(* CODESYS project 0427直角+Delta.project
   CompiledLibraryCompatibilityVersion: LeadSysStudio V3.5 SP15 Patch 4
   Title: Untitled2

Project tree, tasks and I/O mapping:
  Device : PMC600, Leadshine Technology Co., Ltd., order no. 600101, version 3.5.15.40
    application Application
      libraries: Standard, * (System)
      task MainTask (cyclic, interval t#4ms, priority 4, watchdog t#5000ms x 1) calls nothing
      task EtherCAT_Master_Leadshine_A (cyclic, interval 4000 µs, priority 0) calls PLC_PRG, EtherCAT_Master_Leadshine_A.EtherCAT_Task
      task SoftMotion_PlanningTask (freewheeling, priority 15) calls nothing
      program PLC_PRG [LD]
      axis group Tripod: TRAFO.Kin_Tripod_Rotary, axes Axis_3, Axis_4, Axis_5
    Device Diagnose
    Network Configuration
      LocalBus Config
    Resource Usage
    SoftMotion General Axis Pool
    High_Speed_IO_Module : High Speed IO Module, Leadshine Technology Co., Ltd., version 3.5.15.40
        settings: HS counter 2.Counter_Channel = 1; HS counter 3.Counter_Channel = 2; HS counter 4.Counter_Channel = 3; HS counter 5.Counter_Channel = 4; HS counter 6.Counter_Channel = 5
        unmapped channels: Genral_IO_IN, Genral_IO_Out
    EtherCAT_Master_Leadshine_A : EtherCAT Master Leadshine, Leadshine Technology Co., Ltd., version 3.5.9.50
        settings: MasterCycleTime = 4000
      PM32EC_LOCAL : PM32EC-LOCAL, Leadshine Technology Co., Ltd., order no. PM32EC-LOCAL, version Revision=16#20061010
          settings: StationAlias = 0; DC sync0 cycletime = 4000; DC sync1 cycletime = 4000
      DM3C_EC522 : DM3C-EC522(COE), Leadshine Technology Co.,Ltd., order no. DM3C-EC522, version Revision=16#00000001
          settings: StationAlias = 0; DC sync0 cycletime = 4000; DC sync1 cycletime = 4000; Number of SDO = 6; Homing method.Index = 16#6098; Homing method.Subindex = 16#00; Homing method.Value = 17; Homing method.Size = 8; Homing method.AbortIfError = FALSE; Homing method.JumpToLine = FALSE; Homing method.Line = 0; Homing method.CompleteAccess = FALSE; Homing velocity (fast).Index = 16#6099; Homing velocity (fast).Subindex = 16#01; Homing velocity (fast).Value = 16667; Homing velocity (fast).Size = 32; Homing velocity (fast).AbortIfError = FALSE; Homing velocity (fast).JumpToLine = FALSE; Homing velocity (fast).Line = 0; Homing velocity (fast).CompleteAccess = FALSE; Homing velocity (slow).Index = 16#6099; Homing velocity (slow).Subindex = 16#02; Homing velocity (slow).Value = 3333; Homing velocity (slow).Size = 32; Homing velocity (slow).AbortIfError = FALSE; Homing velocity (slow).JumpToLine = FALSE; Homing velocity (slow).Line = 0; Homing velocity (slow).CompleteAccess = FALSE; Homing acceleration.Index = 16#609A; Homing acceleration.Subindex = 16#00; Homing acceleration.Value = 83333; Homing acceleration.Size = 32; Homing acceleration.AbortIfError = FALSE; Homing acceleration.JumpToLine = FALSE; Homing acceleration.Line = 0; Homing acceleration.CompleteAccess = FALSE; Homing offset.Index = 16#607C; Homing offset.Subindex = 16#00; Homing offset.Value = 0; Homing offset.Size = 32;
            Homing offset.AbortIfError = FALSE; Homing offset.JumpToLine = FALSE; Homing offset.Line = 0; Homing offset.CompleteAccess = FALSE
          unmapped channels: Control Word, Profile Target Position, Touch Probe Function, Last Error Code, Status Word, Modes of Operation display, Position Actual Value, Touch Probe Status, Touch Probe 1 Positive Value, Digital Inputs
        Axis : Axis, 3S - Smart Software Solutions GmbH, order no. 0, version 4.6.1.0
            settings: wDriveID = 0; dwRatioTechUnitsDenom = 2500; iRatioTechUnitsNum = 3; 一圈脉冲数 = 50000; 工作台一圈的位移 = 60; 电子齿轮比分子 = 1; 电子齿轮比分母 = 1; ScalingIncs = 2500; ScalingUnits = 3; AdrOffset_8010 = 4; BitOffset_8010 = 0; BitLength_8010 = 16; Address_8010 = '%QW2'; Type_8010 = 'UINT'; AddressPointer_8010 = ADR(%QW2); AdrOffset_8020 = 8; BitOffset_8020 = 0; BitLength_8020 = 32; Address_8020 = '%QD2'; Type_8020 = 'DINT'; AddressPointer_8020 = ADR(%QD2); AdrOffset_8030 = 4294967295; BitOffset_8030 = 0; BitLength_8030 = 32; Address_8030 = ''; Type_8030 = 'DINT'; AddressPointer_8030 = 0; AdrOffset_8040 = 4294967295; BitOffset_8040 = 0; BitLength_8040 = 0; Address_8040 = ''; Type_8040 = ''; AddressPointer_8040 = 0; AdrOffset_8050 = 4294967295; BitOffset_8050 = 0; BitLength_8050 = 8; Address_8050 = ''; Type_8050 = 'USINT'; AddressPointer_8050 = 0; AdrOffset_8060 = 12;
              BitOffset_8060 = 0; BitLength_8060 = 16; Address_8060 = '%QW6'; Type_8060 = 'UINT'; AddressPointer_8060 = ADR(%QW6); AdrOffset_8070 = 4294967295; BitOffset_8070 = 0; BitLength_8070 = 0; Address_8070 = ''; Type_8070 = ''; AddressPointer_8070 = 0; AdrOffset_8080 = 4294967295; BitOffset_8080 = 0; BitLength_8080 = 0; Address_8080 = ''; Type_8080 = ''; AddressPointer_8080 = 0; AdrOffset_8090 = 4294967295; BitOffset_8090 = 0; BitLength_8090 = 0; Address_8090 = ''; Type_8090 = ''; AddressPointer_8090 = 0; AdrOffset_8510 = 6; BitOffset_8510 = 0; BitLength_8510 = 16; Address_8510 = '%IW3'; Type_8510 = 'UINT'; AddressPointer_8510 = ADR(%IW3); AdrOffset_8520 = 12; BitOffset_8520 = 0; BitLength_8520 = 32; Address_8520 = '%ID3'; Type_8520 = 'DINT'; AddressPointer_8520 = ADR(%ID3); AdrOffset_8530 = 4294967295; BitOffset_8530 = 0; BitLength_8530 = 0; Address_8530 = ''; Type_8530 = '';
              AddressPointer_8530 = 0; AdrOffset_8540 = 4294967295; BitOffset_8540 = 0; BitLength_8540 = 0; Address_8540 = ''; Type_8540 = ''; AddressPointer_8540 = 0; AdrOffset_8550 = 8; BitOffset_8550 = 0; BitLength_8550 = 8; Address_8550 = '%IB8'; Type_8550 = 'SINT'; AddressPointer_8550 = ADR(%IB8); AdrOffset_8560 = 24; BitOffset_8560 = 0; BitLength_8560 = 32; Address_8560 = '%ID6'; Type_8560 = 'UDINT'; AddressPointer_8560 = ADR(%ID6); AdrOffset_8570 = 16; BitOffset_8570 = 0; BitLength_8570 = 16; Address_8570 = '%IW8'; Type_8570 = 'UINT'; AddressPointer_8570 = ADR(%IW8); AdrOffset_8580 = 20; BitOffset_8580 = 0; BitLength_8580 = 32; Address_8580 = '%ID5'; Type_8580 = 'DINT'; AddressPointer_8580 = ADR(%ID5); AdrOffset_8590 = 4294967295; BitOffset_8590 = 0; BitLength_8590 = 0; Address_8590 = ''; Type_8590 = ''; AddressPointer_8590 = 0; AdrOffset_8600 = 4294967295; BitOffset_8600 = 0; BitLength_8600 = 0;
              Address_8600 = ''; Type_8600 = ''; AddressPointer_8600 = 0; AdrOffset_8600 = 4294967295; BitOffset_8600 = 0; BitLength_8600 = 0; Address_8610 = ''; Type_8610 = ''; AddressPointer_8610 = 0; AdrOffset_8620 = 4294967295; BitOffset_8620 = 0; BitLength_8620 = 0; Address_8620 = ''; Type_8620 = ''; AddressPointer_8620 = 0
      DM3C_EC522_1 : DM3C-EC522(COE), Leadshine Technology Co.,Ltd., order no. DM3C-EC522, version Revision=16#00000001
          settings: StationAlias = 0; DC sync0 cycletime = 4000; DC sync1 cycletime = 4000; Number of SDO = 6; Homing method.Index = 16#6098; Homing method.Subindex = 16#00; Homing method.Value = 17; Homing method.Size = 8; Homing method.AbortIfError = FALSE; Homing method.JumpToLine = FALSE; Homing method.Line = 0; Homing method.CompleteAccess = FALSE; Homing velocity (fast).Index = 16#6099; Homing velocity (fast).Subindex = 16#01; Homing velocity (fast).Value = 16667; Homing velocity (fast).Size = 32; Homing velocity (fast).AbortIfError = FALSE; Homing velocity (fast).JumpToLine = FALSE; Homing velocity (fast).Line = 0; Homing velocity (fast).CompleteAccess = FALSE; Homing velocity (slow).Index = 16#6099; Homing velocity (slow).Subindex = 16#02; Homing velocity (slow).Value = 3333; Homing velocity (slow).Size = 32; Homing velocity (slow).AbortIfError = FALSE; Homing velocity (slow).JumpToLine = FALSE; Homing velocity (slow).Line = 0; Homing velocity (slow).CompleteAccess = FALSE; Homing acceleration.Index = 16#609A; Homing acceleration.Subindex = 16#00; Homing acceleration.Value = 83333; Homing acceleration.Size = 32; Homing acceleration.AbortIfError = FALSE; Homing acceleration.JumpToLine = FALSE; Homing acceleration.Line = 0; Homing acceleration.CompleteAccess = FALSE; Homing offset.Index = 16#607C; Homing offset.Subindex = 16#00; Homing offset.Value = 0; Homing offset.Size = 32;
            Homing offset.AbortIfError = FALSE; Homing offset.JumpToLine = FALSE; Homing offset.Line = 0; Homing offset.CompleteAccess = FALSE
          unmapped channels: Control Word, Profile Target Position, Touch Probe Function, Last Error Code, Status Word, Modes of Operation display, Position Actual Value, Touch Probe Status, Touch Probe 1 Positive Value, Digital Inputs
        Axis_1 : Axis, 3S - Smart Software Solutions GmbH, order no. 0, version 4.6.1.0
            settings: dwRatioTechUnitsDenom = 2500; iRatioTechUnitsNum = 3; 一圈脉冲数 = 50000; 工作台一圈的位移 = 60; 电子齿轮比分子 = 1; 电子齿轮比分母 = 1; ScalingIncs = 2500; ScalingUnits = 3; AdrOffset_8010 = 16; BitOffset_8010 = 0; BitLength_8010 = 16; Address_8010 = '%QW8'; Type_8010 = 'UINT'; AddressPointer_8010 = ADR(%QW8); AdrOffset_8020 = 20; BitOffset_8020 = 0; BitLength_8020 = 32; Address_8020 = '%QD5'; Type_8020 = 'DINT'; AddressPointer_8020 = ADR(%QD5); AdrOffset_8030 = 4294967295; BitOffset_8030 = 0; BitLength_8030 = 32; Address_8030 = ''; Type_8030 = 'DINT'; AddressPointer_8030 = 0; AdrOffset_8040 = 4294967295; BitOffset_8040 = 0; BitLength_8040 = 0; Address_8040 = ''; Type_8040 = ''; AddressPointer_8040 = 0; AdrOffset_8050 = 4294967295; BitOffset_8050 = 0; BitLength_8050 = 8; Address_8050 = ''; Type_8050 = 'USINT'; AddressPointer_8050 = 0; AdrOffset_8060 = 24; BitOffset_8060 = 0;
              BitLength_8060 = 16; Address_8060 = '%QW12'; Type_8060 = 'UINT'; AddressPointer_8060 = ADR(%QW12); AdrOffset_8070 = 4294967295; BitOffset_8070 = 0; BitLength_8070 = 0; Address_8070 = ''; Type_8070 = ''; AddressPointer_8070 = 0; AdrOffset_8080 = 4294967295; BitOffset_8080 = 0; BitLength_8080 = 0; Address_8080 = ''; Type_8080 = ''; AddressPointer_8080 = 0; AdrOffset_8090 = 4294967295; BitOffset_8090 = 0; BitLength_8090 = 0; Address_8090 = ''; Type_8090 = ''; AddressPointer_8090 = 0; AdrOffset_8510 = 30; BitOffset_8510 = 0; BitLength_8510 = 16; Address_8510 = '%IW15'; Type_8510 = 'UINT'; AddressPointer_8510 = ADR(%IW15); AdrOffset_8520 = 36; BitOffset_8520 = 0; BitLength_8520 = 32; Address_8520 = '%ID9'; Type_8520 = 'DINT'; AddressPointer_8520 = ADR(%ID9); AdrOffset_8530 = 4294967295; BitOffset_8530 = 0; BitLength_8530 = 0; Address_8530 = ''; Type_8530 = ''; AddressPointer_8530 = 0;
              AdrOffset_8540 = 4294967295; BitOffset_8540 = 0; BitLength_8540 = 0; Address_8540 = ''; Type_8540 = ''; AddressPointer_8540 = 0; AdrOffset_8550 = 32; BitOffset_8550 = 0; BitLength_8550 = 8; Address_8550 = '%IB32'; Type_8550 = 'SINT'; AddressPointer_8550 = ADR(%IB32); AdrOffset_8560 = 48; BitOffset_8560 = 0; BitLength_8560 = 32; Address_8560 = '%ID12'; Type_8560 = 'UDINT'; AddressPointer_8560 = ADR(%ID12); AdrOffset_8570 = 40; BitOffset_8570 = 0; BitLength_8570 = 16; Address_8570 = '%IW20'; Type_8570 = 'UINT'; AddressPointer_8570 = ADR(%IW20); AdrOffset_8580 = 44; BitOffset_8580 = 0; BitLength_8580 = 32; Address_8580 = '%ID11'; Type_8580 = 'DINT'; AddressPointer_8580 = ADR(%ID11); AdrOffset_8590 = 4294967295; BitOffset_8590 = 0; BitLength_8590 = 0; Address_8590 = ''; Type_8590 = ''; AddressPointer_8590 = 0; AdrOffset_8600 = 4294967295; BitOffset_8600 = 0; BitLength_8600 = 0; Address_8600 = '';
              Type_8600 = ''; AddressPointer_8600 = 0; AdrOffset_8600 = 4294967295; BitOffset_8600 = 0; BitLength_8600 = 0; Address_8610 = ''; Type_8610 = ''; AddressPointer_8610 = 0; AdrOffset_8620 = 4294967295; BitOffset_8620 = 0; BitLength_8620 = 0; Address_8620 = ''; Type_8620 = ''; AddressPointer_8620 = 0
      DM3C_EC522_2 : DM3C-EC522(COE), Leadshine Technology Co.,Ltd., order no. DM3C-EC522, version Revision=16#00000001
          settings: StationAlias = 0; DC sync0 cycletime = 4000; DC sync1 cycletime = 4000; Number of SDO = 6; Homing method.Index = 16#6098; Homing method.Subindex = 16#00; Homing method.Value = 17; Homing method.Size = 8; Homing method.AbortIfError = FALSE; Homing method.JumpToLine = FALSE; Homing method.Line = 0; Homing method.CompleteAccess = FALSE; Homing velocity (fast).Index = 16#6099; Homing velocity (fast).Subindex = 16#01; Homing velocity (fast).Value = 125000; Homing velocity (fast).Size = 32; Homing velocity (fast).AbortIfError = FALSE; Homing velocity (fast).JumpToLine = FALSE; Homing velocity (fast).Line = 0; Homing velocity (fast).CompleteAccess = FALSE; Homing velocity (slow).Index = 16#6099; Homing velocity (slow).Subindex = 16#02; Homing velocity (slow).Value = 25000; Homing velocity (slow).Size = 32; Homing velocity (slow).AbortIfError = FALSE; Homing velocity (slow).JumpToLine = FALSE; Homing velocity (slow).Line = 0; Homing velocity (slow).CompleteAccess = FALSE; Homing acceleration.Index = 16#609A; Homing acceleration.Subindex = 16#00; Homing acceleration.Value = 1250000; Homing acceleration.Size = 32; Homing acceleration.AbortIfError = FALSE; Homing acceleration.JumpToLine = FALSE; Homing acceleration.Line = 0; Homing acceleration.CompleteAccess = FALSE; Homing offset.Index = 16#607C; Homing offset.Subindex = 16#00; Homing offset.Value = 0; Homing offset.Size = 32;
            Homing offset.AbortIfError = FALSE; Homing offset.JumpToLine = FALSE; Homing offset.Line = 0; Homing offset.CompleteAccess = FALSE
          unmapped channels: Control Word, Profile Target Position, Touch Probe Function, Last Error Code, Status Word, Modes of Operation display, Position Actual Value, Touch Probe Status, Touch Probe 1 Positive Value, Digital Inputs
        Axis_2 : Axis, 3S - Smart Software Solutions GmbH, order no. 0, version 4.6.1.0
            settings: wDriveID = 2; dwRatioTechUnitsDenom = 12500; 一圈脉冲数 = 50000; 工作台一圈的位移 = 4; 电子齿轮比分子 = 1; 电子齿轮比分母 = 1; ScalingIncs = 12500; AdrOffset_8010 = 28; BitOffset_8010 = 0; BitLength_8010 = 16; Address_8010 = '%QW14'; Type_8010 = 'UINT'; AddressPointer_8010 = ADR(%QW14); AdrOffset_8020 = 32; BitOffset_8020 = 0; BitLength_8020 = 32; Address_8020 = '%QD8'; Type_8020 = 'DINT'; AddressPointer_8020 = ADR(%QD8); AdrOffset_8030 = 4294967295; BitOffset_8030 = 0; BitLength_8030 = 32; Address_8030 = ''; Type_8030 = 'DINT'; AddressPointer_8030 = 0; AdrOffset_8040 = 4294967295; BitOffset_8040 = 0; BitLength_8040 = 0; Address_8040 = ''; Type_8040 = ''; AddressPointer_8040 = 0; AdrOffset_8050 = 4294967295; BitOffset_8050 = 0; BitLength_8050 = 8; Address_8050 = ''; Type_8050 = 'USINT'; AddressPointer_8050 = 0; AdrOffset_8060 = 36; BitOffset_8060 = 0; BitLength_8060 = 16;
              Address_8060 = '%QW18'; Type_8060 = 'UINT'; AddressPointer_8060 = ADR(%QW18); AdrOffset_8070 = 4294967295; BitOffset_8070 = 0; BitLength_8070 = 0; Address_8070 = ''; Type_8070 = ''; AddressPointer_8070 = 0; AdrOffset_8080 = 4294967295; BitOffset_8080 = 0; BitLength_8080 = 0; Address_8080 = ''; Type_8080 = ''; AddressPointer_8080 = 0; AdrOffset_8090 = 4294967295; BitOffset_8090 = 0; BitLength_8090 = 0; Address_8090 = ''; Type_8090 = ''; AddressPointer_8090 = 0; AdrOffset_8510 = 54; BitOffset_8510 = 0; BitLength_8510 = 16; Address_8510 = '%IW27'; Type_8510 = 'UINT'; AddressPointer_8510 = ADR(%IW27); AdrOffset_8520 = 60; BitOffset_8520 = 0; BitLength_8520 = 32; Address_8520 = '%ID15'; Type_8520 = 'DINT'; AddressPointer_8520 = ADR(%ID15); AdrOffset_8530 = 4294967295; BitOffset_8530 = 0; BitLength_8530 = 0; Address_8530 = ''; Type_8530 = ''; AddressPointer_8530 = 0; AdrOffset_8540 = 4294967295;
              BitOffset_8540 = 0; BitLength_8540 = 0; Address_8540 = ''; Type_8540 = ''; AddressPointer_8540 = 0; AdrOffset_8550 = 56; BitOffset_8550 = 0; BitLength_8550 = 8; Address_8550 = '%IB56'; Type_8550 = 'SINT'; AddressPointer_8550 = ADR(%IB56); AdrOffset_8560 = 72; BitOffset_8560 = 0; BitLength_8560 = 32; Address_8560 = '%ID18'; Type_8560 = 'UDINT'; AddressPointer_8560 = ADR(%ID18); AdrOffset_8570 = 64; BitOffset_8570 = 0; BitLength_8570 = 16; Address_8570 = '%IW32'; Type_8570 = 'UINT'; AddressPointer_8570 = ADR(%IW32); AdrOffset_8580 = 68; BitOffset_8580 = 0; BitLength_8580 = 32; Address_8580 = '%ID17'; Type_8580 = 'DINT'; AddressPointer_8580 = ADR(%ID17); AdrOffset_8590 = 4294967295; BitOffset_8590 = 0; BitLength_8590 = 0; Address_8590 = ''; Type_8590 = ''; AddressPointer_8590 = 0; AdrOffset_8600 = 4294967295; BitOffset_8600 = 0; BitLength_8600 = 0; Address_8600 = ''; Type_8600 = '';
              AddressPointer_8600 = 0; AdrOffset_8600 = 4294967295; BitOffset_8600 = 0; BitLength_8600 = 0; Address_8610 = ''; Type_8610 = ''; AddressPointer_8610 = 0; AdrOffset_8620 = 4294967295; BitOffset_8620 = 0; BitLength_8620 = 0; Address_8620 = ''; Type_8620 = ''; AddressPointer_8620 = 0
      DM3C_EC522_3 : DM3C-EC522(COE), Leadshine Technology Co.,Ltd., order no. DM3C-EC522, version Revision=16#00000001
          settings: StationAlias = 0; DC sync0 cycletime = 4000; DC sync1 cycletime = 4000; Number of SDO = 6; Homing method.Index = 16#6098; Homing method.Subindex = 16#00; Homing method.Value = 21; Homing method.Size = 8; Homing method.AbortIfError = FALSE; Homing method.JumpToLine = FALSE; Homing method.Line = 0; Homing method.CompleteAccess = FALSE; Homing velocity (fast).Index = 16#6099; Homing velocity (fast).Subindex = 16#01; Homing velocity (fast).Value = 7500; Homing velocity (fast).Size = 32; Homing velocity (fast).AbortIfError = FALSE; Homing velocity (fast).JumpToLine = FALSE; Homing velocity (fast).Line = 0; Homing velocity (fast).CompleteAccess = FALSE; Homing velocity (slow).Index = 16#6099; Homing velocity (slow).Subindex = 16#02; Homing velocity (slow).Value = 1500; Homing velocity (slow).Size = 32; Homing velocity (slow).AbortIfError = FALSE; Homing velocity (slow).JumpToLine = FALSE; Homing velocity (slow).Line = 0; Homing velocity (slow).CompleteAccess = FALSE; Homing acceleration.Index = 16#609A; Homing acceleration.Subindex = 16#00; Homing acceleration.Value = 50000; Homing acceleration.Size = 32; Homing acceleration.AbortIfError = FALSE; Homing acceleration.JumpToLine = FALSE; Homing acceleration.Line = 0; Homing acceleration.CompleteAccess = FALSE; Homing offset.Index = 16#607C; Homing offset.Subindex = 16#00; Homing offset.Value = 0; Homing offset.Size = 32;
            Homing offset.AbortIfError = FALSE; Homing offset.JumpToLine = FALSE; Homing offset.Line = 0; Homing offset.CompleteAccess = FALSE
          unmapped channels: Control Word, Profile Target Position, Touch Probe Function, Last Error Code, Status Word, Modes of Operation display, Position Actual Value, Touch Probe Status, Touch Probe 1 Positive Value, Digital Inputs
        Axis_3 : Axis, 3S - Smart Software Solutions GmbH, order no. 0, version 4.6.1.0
            settings: wDriveID = 3; dwRatioTechUnitsDenom = 500; iRatioTechUnitsNum = -1; 一圈脉冲数 = 36000; 工作台一圈的位移 = 360; 电子齿轮比分子 = 5; 电子齿轮比分母 = 1; ScalingIncs = 500; InvertDirection = True; AdrOffset_8010 = 40; BitOffset_8010 = 0; BitLength_8010 = 16; Address_8010 = '%QW20'; Type_8010 = 'UINT'; AddressPointer_8010 = ADR(%QW20); AdrOffset_8020 = 44; BitOffset_8020 = 0; BitLength_8020 = 32; Address_8020 = '%QD11'; Type_8020 = 'DINT'; AddressPointer_8020 = ADR(%QD11); AdrOffset_8030 = 4294967295; BitOffset_8030 = 0; BitLength_8030 = 32; Address_8030 = ''; Type_8030 = 'DINT'; AddressPointer_8030 = 0; AdrOffset_8040 = 4294967295; BitOffset_8040 = 0; BitLength_8040 = 0; Address_8040 = ''; Type_8040 = ''; AddressPointer_8040 = 0; AdrOffset_8050 = 4294967295; BitOffset_8050 = 0; BitLength_8050 = 8; Address_8050 = ''; Type_8050 = 'USINT'; AddressPointer_8050 = 0; AdrOffset_8060 = 48;
              BitOffset_8060 = 0; BitLength_8060 = 16; Address_8060 = '%QW24'; Type_8060 = 'UINT'; AddressPointer_8060 = ADR(%QW24); AdrOffset_8070 = 4294967295; BitOffset_8070 = 0; BitLength_8070 = 0; Address_8070 = ''; Type_8070 = ''; AddressPointer_8070 = 0; AdrOffset_8080 = 4294967295; BitOffset_8080 = 0; BitLength_8080 = 0; Address_8080 = ''; Type_8080 = ''; AddressPointer_8080 = 0; AdrOffset_8090 = 4294967295; BitOffset_8090 = 0; BitLength_8090 = 0; Address_8090 = ''; Type_8090 = ''; AddressPointer_8090 = 0; AdrOffset_8510 = 78; BitOffset_8510 = 0; BitLength_8510 = 16; Address_8510 = '%IW39'; Type_8510 = 'UINT'; AddressPointer_8510 = ADR(%IW39); AdrOffset_8520 = 84; BitOffset_8520 = 0; BitLength_8520 = 32; Address_8520 = '%ID21'; Type_8520 = 'DINT'; AddressPointer_8520 = ADR(%ID21); AdrOffset_8530 = 4294967295; BitOffset_8530 = 0; BitLength_8530 = 0; Address_8530 = ''; Type_8530 = '';
              AddressPointer_8530 = 0; AdrOffset_8540 = 4294967295; BitOffset_8540 = 0; BitLength_8540 = 0; Address_8540 = ''; Type_8540 = ''; AddressPointer_8540 = 0; AdrOffset_8550 = 80; BitOffset_8550 = 0; BitLength_8550 = 8; Address_8550 = '%IB80'; Type_8550 = 'SINT'; AddressPointer_8550 = ADR(%IB80); AdrOffset_8560 = 96; BitOffset_8560 = 0; BitLength_8560 = 32; Address_8560 = '%ID24'; Type_8560 = 'UDINT'; AddressPointer_8560 = ADR(%ID24); AdrOffset_8570 = 88; BitOffset_8570 = 0; BitLength_8570 = 16; Address_8570 = '%IW44'; Type_8570 = 'UINT'; AddressPointer_8570 = ADR(%IW44); AdrOffset_8580 = 92; BitOffset_8580 = 0; BitLength_8580 = 32; Address_8580 = '%ID23'; Type_8580 = 'DINT'; AddressPointer_8580 = ADR(%ID23); AdrOffset_8590 = 4294967295; BitOffset_8590 = 0; BitLength_8590 = 0; Address_8590 = ''; Type_8590 = ''; AddressPointer_8590 = 0; AdrOffset_8600 = 4294967295; BitOffset_8600 = 0; BitLength_8600 = 0;
              Address_8600 = ''; Type_8600 = ''; AddressPointer_8600 = 0; AdrOffset_8600 = 4294967295; BitOffset_8600 = 0; BitLength_8600 = 0; Address_8610 = ''; Type_8610 = ''; AddressPointer_8610 = 0; AdrOffset_8620 = 4294967295; BitOffset_8620 = 0; BitLength_8620 = 0; Address_8620 = ''; Type_8620 = ''; AddressPointer_8620 = 0
      DM3C_EC522_4 : DM3C-EC522(COE), Leadshine Technology Co.,Ltd., order no. DM3C-EC522, version Revision=16#00000001
          settings: StationAlias = 0; DC sync0 cycletime = 4000; DC sync1 cycletime = 4000; Number of SDO = 6; Homing method.Index = 16#6098; Homing method.Subindex = 16#00; Homing method.Value = 21; Homing method.Size = 8; Homing method.AbortIfError = FALSE; Homing method.JumpToLine = FALSE; Homing method.Line = 0; Homing method.CompleteAccess = FALSE; Homing velocity (fast).Index = 16#6099; Homing velocity (fast).Subindex = 16#01; Homing velocity (fast).Value = 7500; Homing velocity (fast).Size = 32; Homing velocity (fast).AbortIfError = FALSE; Homing velocity (fast).JumpToLine = FALSE; Homing velocity (fast).Line = 0; Homing velocity (fast).CompleteAccess = FALSE; Homing velocity (slow).Index = 16#6099; Homing velocity (slow).Subindex = 16#02; Homing velocity (slow).Value = 1500; Homing velocity (slow).Size = 32; Homing velocity (slow).AbortIfError = FALSE; Homing velocity (slow).JumpToLine = FALSE; Homing velocity (slow).Line = 0; Homing velocity (slow).CompleteAccess = FALSE; Homing acceleration.Index = 16#609A; Homing acceleration.Subindex = 16#00; Homing acceleration.Value = 50000; Homing acceleration.Size = 32; Homing acceleration.AbortIfError = FALSE; Homing acceleration.JumpToLine = FALSE; Homing acceleration.Line = 0; Homing acceleration.CompleteAccess = FALSE; Homing offset.Index = 16#607C; Homing offset.Subindex = 16#00; Homing offset.Value = 0; Homing offset.Size = 32;
            Homing offset.AbortIfError = FALSE; Homing offset.JumpToLine = FALSE; Homing offset.Line = 0; Homing offset.CompleteAccess = FALSE
          unmapped channels: Control Word, Profile Target Position, Touch Probe Function, Last Error Code, Status Word, Modes of Operation display, Position Actual Value, Touch Probe Status, Touch Probe 1 Positive Value, Digital Inputs
        Axis_4 : Axis, 3S - Smart Software Solutions GmbH, order no. 0, version 4.6.1.0
            settings: wDriveID = 4; dwRatioTechUnitsDenom = 500; iRatioTechUnitsNum = -1; 一圈脉冲数 = 36000; 工作台一圈的位移 = 360; 电子齿轮比分子 = 5; 电子齿轮比分母 = 1; ScalingIncs = 500; InvertDirection = True; AdrOffset_8010 = 52; BitOffset_8010 = 0; BitLength_8010 = 16; Address_8010 = '%QW26'; Type_8010 = 'UINT'; AddressPointer_8010 = ADR(%QW26); AdrOffset_8020 = 56; BitOffset_8020 = 0; BitLength_8020 = 32; Address_8020 = '%QD14'; Type_8020 = 'DINT'; AddressPointer_8020 = ADR(%QD14); AdrOffset_8030 = 4294967295; BitOffset_8030 = 0; BitLength_8030 = 32; Address_8030 = ''; Type_8030 = 'DINT'; AddressPointer_8030 = 0; AdrOffset_8040 = 4294967295; BitOffset_8040 = 0; BitLength_8040 = 0; Address_8040 = ''; Type_8040 = ''; AddressPointer_8040 = 0; AdrOffset_8050 = 4294967295; BitOffset_8050 = 0; BitLength_8050 = 8; Address_8050 = ''; Type_8050 = 'USINT'; AddressPointer_8050 = 0; AdrOffset_8060 = 60;
              BitOffset_8060 = 0; BitLength_8060 = 16; Address_8060 = '%QW30'; Type_8060 = 'UINT'; AddressPointer_8060 = ADR(%QW30); AdrOffset_8070 = 4294967295; BitOffset_8070 = 0; BitLength_8070 = 0; Address_8070 = ''; Type_8070 = ''; AddressPointer_8070 = 0; AdrOffset_8080 = 4294967295; BitOffset_8080 = 0; BitLength_8080 = 0; Address_8080 = ''; Type_8080 = ''; AddressPointer_8080 = 0; AdrOffset_8090 = 4294967295; BitOffset_8090 = 0; BitLength_8090 = 0; Address_8090 = ''; Type_8090 = ''; AddressPointer_8090 = 0; AdrOffset_8510 = 102; BitOffset_8510 = 0; BitLength_8510 = 16; Address_8510 = '%IW51'; Type_8510 = 'UINT'; AddressPointer_8510 = ADR(%IW51); AdrOffset_8520 = 108; BitOffset_8520 = 0; BitLength_8520 = 32; Address_8520 = '%ID27'; Type_8520 = 'DINT'; AddressPointer_8520 = ADR(%ID27); AdrOffset_8530 = 4294967295; BitOffset_8530 = 0; BitLength_8530 = 0; Address_8530 = ''; Type_8530 = '';
              AddressPointer_8530 = 0; AdrOffset_8540 = 4294967295; BitOffset_8540 = 0; BitLength_8540 = 0; Address_8540 = ''; Type_8540 = ''; AddressPointer_8540 = 0; AdrOffset_8550 = 104; BitOffset_8550 = 0; BitLength_8550 = 8; Address_8550 = '%IB104'; Type_8550 = 'SINT'; AddressPointer_8550 = ADR(%IB104); AdrOffset_8560 = 120; BitOffset_8560 = 0; BitLength_8560 = 32; Address_8560 = '%ID30'; Type_8560 = 'UDINT'; AddressPointer_8560 = ADR(%ID30); AdrOffset_8570 = 112; BitOffset_8570 = 0; BitLength_8570 = 16; Address_8570 = '%IW56'; Type_8570 = 'UINT'; AddressPointer_8570 = ADR(%IW56); AdrOffset_8580 = 116; BitOffset_8580 = 0; BitLength_8580 = 32; Address_8580 = '%ID29'; Type_8580 = 'DINT'; AddressPointer_8580 = ADR(%ID29); AdrOffset_8590 = 4294967295; BitOffset_8590 = 0; BitLength_8590 = 0; Address_8590 = ''; Type_8590 = ''; AddressPointer_8590 = 0; AdrOffset_8600 = 4294967295; BitOffset_8600 = 0; BitLength_8600 = 0;
              Address_8600 = ''; Type_8600 = ''; AddressPointer_8600 = 0; AdrOffset_8600 = 4294967295; BitOffset_8600 = 0; BitLength_8600 = 0; Address_8610 = ''; Type_8610 = ''; AddressPointer_8610 = 0; AdrOffset_8620 = 4294967295; BitOffset_8620 = 0; BitLength_8620 = 0; Address_8620 = ''; Type_8620 = ''; AddressPointer_8620 = 0
      DM3C_EC522_5 : DM3C-EC522(COE), Leadshine Technology Co.,Ltd., order no. DM3C-EC522, version Revision=16#00000001
          settings: StationAlias = 0; DC sync0 cycletime = 4000; DC sync1 cycletime = 4000; Number of SDO = 6; Homing method.Index = 16#6098; Homing method.Subindex = 16#00; Homing method.Value = 21; Homing method.Size = 8; Homing method.AbortIfError = FALSE; Homing method.JumpToLine = FALSE; Homing method.Line = 0; Homing method.CompleteAccess = FALSE; Homing velocity (fast).Index = 16#6099; Homing velocity (fast).Subindex = 16#01; Homing velocity (fast).Value = 7500; Homing velocity (fast).Size = 32; Homing velocity (fast).AbortIfError = FALSE; Homing velocity (fast).JumpToLine = FALSE; Homing velocity (fast).Line = 0; Homing velocity (fast).CompleteAccess = FALSE; Homing velocity (slow).Index = 16#6099; Homing velocity (slow).Subindex = 16#02; Homing velocity (slow).Value = 1500; Homing velocity (slow).Size = 32; Homing velocity (slow).AbortIfError = FALSE; Homing velocity (slow).JumpToLine = FALSE; Homing velocity (slow).Line = 0; Homing velocity (slow).CompleteAccess = FALSE; Homing acceleration.Index = 16#609A; Homing acceleration.Subindex = 16#00; Homing acceleration.Value = 50000; Homing acceleration.Size = 32; Homing acceleration.AbortIfError = FALSE; Homing acceleration.JumpToLine = FALSE; Homing acceleration.Line = 0; Homing acceleration.CompleteAccess = FALSE; Homing offset.Index = 16#607C; Homing offset.Subindex = 16#00; Homing offset.Value = 0; Homing offset.Size = 32;
            Homing offset.AbortIfError = FALSE; Homing offset.JumpToLine = FALSE; Homing offset.Line = 0; Homing offset.CompleteAccess = FALSE
          unmapped channels: Control Word, Profile Target Position, Touch Probe Function, Last Error Code, Status Word, Modes of Operation display, Position Actual Value, Touch Probe Status, Touch Probe 1 Positive Value, Digital Inputs
        Axis_5 : Axis, 3S - Smart Software Solutions GmbH, order no. 0, version 4.6.1.0
            settings: wDriveID = 5; dwRatioTechUnitsDenom = 500; iRatioTechUnitsNum = -1; 一圈脉冲数 = 36000; 工作台一圈的位移 = 360; 电子齿轮比分子 = 5; 电子齿轮比分母 = 1; ScalingIncs = 500; InvertDirection = True; AdrOffset_8010 = 64; BitOffset_8010 = 0; BitLength_8010 = 16; Address_8010 = '%QW32'; Type_8010 = 'UINT'; AddressPointer_8010 = ADR(%QW32); AdrOffset_8020 = 68; BitOffset_8020 = 0; BitLength_8020 = 32; Address_8020 = '%QD17'; Type_8020 = 'DINT'; AddressPointer_8020 = ADR(%QD17); AdrOffset_8030 = 4294967295; BitOffset_8030 = 0; BitLength_8030 = 32; Address_8030 = ''; Type_8030 = 'DINT'; AddressPointer_8030 = 0; AdrOffset_8040 = 4294967295; BitOffset_8040 = 0; BitLength_8040 = 0; Address_8040 = ''; Type_8040 = ''; AddressPointer_8040 = 0; AdrOffset_8050 = 4294967295; BitOffset_8050 = 0; BitLength_8050 = 8; Address_8050 = ''; Type_8050 = 'USINT'; AddressPointer_8050 = 0; AdrOffset_8060 = 72;
              BitOffset_8060 = 0; BitLength_8060 = 16; Address_8060 = '%QW36'; Type_8060 = 'UINT'; AddressPointer_8060 = ADR(%QW36); AdrOffset_8070 = 4294967295; BitOffset_8070 = 0; BitLength_8070 = 0; Address_8070 = ''; Type_8070 = ''; AddressPointer_8070 = 0; AdrOffset_8080 = 4294967295; BitOffset_8080 = 0; BitLength_8080 = 0; Address_8080 = ''; Type_8080 = ''; AddressPointer_8080 = 0; AdrOffset_8090 = 4294967295; BitOffset_8090 = 0; BitLength_8090 = 0; Address_8090 = ''; Type_8090 = ''; AddressPointer_8090 = 0; AdrOffset_8510 = 126; BitOffset_8510 = 0; BitLength_8510 = 16; Address_8510 = '%IW63'; Type_8510 = 'UINT'; AddressPointer_8510 = ADR(%IW63); AdrOffset_8520 = 132; BitOffset_8520 = 0; BitLength_8520 = 32; Address_8520 = '%ID33'; Type_8520 = 'DINT'; AddressPointer_8520 = ADR(%ID33); AdrOffset_8530 = 4294967295; BitOffset_8530 = 0; BitLength_8530 = 0; Address_8530 = ''; Type_8530 = '';
              AddressPointer_8530 = 0; AdrOffset_8540 = 4294967295; BitOffset_8540 = 0; BitLength_8540 = 0; Address_8540 = ''; Type_8540 = ''; AddressPointer_8540 = 0; AdrOffset_8550 = 128; BitOffset_8550 = 0; BitLength_8550 = 8; Address_8550 = '%IB128'; Type_8550 = 'SINT'; AddressPointer_8550 = ADR(%IB128); AdrOffset_8560 = 144; BitOffset_8560 = 0; BitLength_8560 = 32; Address_8560 = '%ID36'; Type_8560 = 'UDINT'; AddressPointer_8560 = ADR(%ID36); AdrOffset_8570 = 136; BitOffset_8570 = 0; BitLength_8570 = 16; Address_8570 = '%IW68'; Type_8570 = 'UINT'; AddressPointer_8570 = ADR(%IW68); AdrOffset_8580 = 140; BitOffset_8580 = 0; BitLength_8580 = 32; Address_8580 = '%ID35'; Type_8580 = 'DINT'; AddressPointer_8580 = ADR(%ID35); AdrOffset_8590 = 4294967295; BitOffset_8590 = 0; BitLength_8590 = 0; Address_8590 = ''; Type_8590 = ''; AddressPointer_8590 = 0; AdrOffset_8600 = 4294967295; BitOffset_8600 = 0; BitLength_8600 = 0;
              Address_8600 = ''; Type_8600 = ''; AddressPointer_8600 = 0; AdrOffset_8600 = 4294967295; BitOffset_8600 = 0; BitLength_8600 = 0; Address_8610 = ''; Type_8610 = ''; AddressPointer_8610 = 0; AdrOffset_8620 = 4294967295; BitOffset_8620 = 0; BitLength_8620 = 0; Address_8620 = ''; Type_8620 = ''; AddressPointer_8620 = 0
      L7EC_100 : L7EC-100(COE), Leadshine Technology Co.,Ltd., order no. L7EC-100, version Revision=16#00000001
          settings: StationAlias = 0; DC sync0 cycletime = 4000; DC sync1 cycletime = 4000; Number of SDO = 6; Homing method.Index = 16#6098; Homing method.Subindex = 16#00; Homing method.Value = 14; Homing method.Size = 8; Homing method.AbortIfError = FALSE; Homing method.JumpToLine = FALSE; Homing method.Line = 0; Homing method.CompleteAccess = FALSE; Homing velocity (fast).Index = 16#6099; Homing velocity (fast).Subindex = 16#01; Homing velocity (fast).Value = 800000; Homing velocity (fast).Size = 32; Homing velocity (fast).AbortIfError = FALSE; Homing velocity (fast).JumpToLine = FALSE; Homing velocity (fast).Line = 0; Homing velocity (fast).CompleteAccess = FALSE; Homing velocity (slow).Index = 16#6099; Homing velocity (slow).Subindex = 16#02; Homing velocity (slow).Value = 48000; Homing velocity (slow).Size = 32; Homing velocity (slow).AbortIfError = FALSE; Homing velocity (slow).JumpToLine = FALSE; Homing velocity (slow).Line = 0; Homing velocity (slow).CompleteAccess = FALSE; Homing acceleration.Index = 16#609A; Homing acceleration.Subindex = 16#00; Homing acceleration.Value = 800000; Homing acceleration.Size = 32; Homing acceleration.AbortIfError = FALSE; Homing acceleration.JumpToLine = FALSE; Homing acceleration.Line = 0; Homing acceleration.CompleteAccess = FALSE; Homing offset.Index = 16#607C; Homing offset.Subindex = 16#00; Homing offset.Value = 0; Homing offset.Size = 32;
            Homing offset.AbortIfError = FALSE; Homing offset.JumpToLine = FALSE; Homing offset.Line = 0; Homing offset.CompleteAccess = FALSE
          unmapped channels: Control word, Profile target position, Touch Probe Function, Last error code, Status word, Modes of operation display, Actual motor position, Touch Probe Status, Touch probe pos1 pos value, Digital inputs
        Axis_6 : Axis, 3S - Smart Software Solutions GmbH, order no. 0, version 4.6.1.0
            settings: wDriveID = 6; dwRatioTechUnitsDenom = 8000; 一圈脉冲数 = 20000; 工作台一圈的位移 = 2.5; 电子齿轮比分子 = 1; 电子齿轮比分母 = 1; ScalingIncs = 8000; AdrOffset_8010 = 76; BitOffset_8010 = 0; BitLength_8010 = 16; Address_8010 = '%QW38'; Type_8010 = 'UINT'; AddressPointer_8010 = ADR(%QW38); AdrOffset_8020 = 80; BitOffset_8020 = 0; BitLength_8020 = 32; Address_8020 = '%QD20'; Type_8020 = 'DINT'; AddressPointer_8020 = ADR(%QD20); AdrOffset_8030 = 4294967295; BitOffset_8030 = 0; BitLength_8030 = 32; Address_8030 = ''; Type_8030 = 'DINT'; AddressPointer_8030 = 0; AdrOffset_8040 = 4294967295; BitOffset_8040 = 0; BitLength_8040 = 16; Address_8040 = ''; Type_8040 = 'INT'; AddressPointer_8040 = 0; AdrOffset_8050 = 4294967295; BitOffset_8050 = 0; BitLength_8050 = 8; Address_8050 = ''; Type_8050 = 'USINT'; AddressPointer_8050 = 0; AdrOffset_8060 = 84; BitOffset_8060 = 0; BitLength_8060 = 16;
              Address_8060 = '%QW42'; Type_8060 = 'UINT'; AddressPointer_8060 = ADR(%QW42); AdrOffset_8070 = 4294967295; BitOffset_8070 = 0; BitLength_8070 = 0; Address_8070 = ''; Type_8070 = ''; AddressPointer_8070 = 0; AdrOffset_8080 = 4294967295; BitOffset_8080 = 0; BitLength_8080 = 16; Address_8080 = ''; Type_8080 = 'INT'; AddressPointer_8080 = 0; AdrOffset_8090 = 4294967295; BitOffset_8090 = 0; BitLength_8090 = 0; Address_8090 = ''; Type_8090 = ''; AddressPointer_8090 = 0; AdrOffset_8510 = 150; BitOffset_8510 = 0; BitLength_8510 = 16; Address_8510 = '%IW75'; Type_8510 = 'UINT'; AddressPointer_8510 = ADR(%IW75); AdrOffset_8520 = 156; BitOffset_8520 = 0; BitLength_8520 = 32; Address_8520 = '%ID39'; Type_8520 = 'DINT'; AddressPointer_8520 = ADR(%ID39); AdrOffset_8530 = 4294967295; BitOffset_8530 = 0; BitLength_8530 = 0; Address_8530 = ''; Type_8530 = ''; AddressPointer_8530 = 0; AdrOffset_8540 = 4294967295;
              BitOffset_8540 = 0; BitLength_8540 = 0; Address_8540 = ''; Type_8540 = ''; AddressPointer_8540 = 0; AdrOffset_8550 = 152; BitOffset_8550 = 0; BitLength_8550 = 8; Address_8550 = '%IB152'; Type_8550 = 'SINT'; AddressPointer_8550 = ADR(%IB152); AdrOffset_8560 = 168; BitOffset_8560 = 0; BitLength_8560 = 32; Address_8560 = '%ID42'; Type_8560 = 'UDINT'; AddressPointer_8560 = ADR(%ID42); AdrOffset_8570 = 160; BitOffset_8570 = 0; BitLength_8570 = 16; Address_8570 = '%IW80'; Type_8570 = 'UINT'; AddressPointer_8570 = ADR(%IW80); AdrOffset_8580 = 164; BitOffset_8580 = 0; BitLength_8580 = 32; Address_8580 = '%ID41'; Type_8580 = 'DINT'; AddressPointer_8580 = ADR(%ID41); AdrOffset_8590 = 4294967295; BitOffset_8590 = 0; BitLength_8590 = 0; Address_8590 = ''; Type_8590 = ''; AddressPointer_8590 = 0; AdrOffset_8600 = 4294967295; BitOffset_8600 = 0; BitLength_8600 = 0; Address_8600 = ''; Type_8600 = '';
              AddressPointer_8600 = 0; AdrOffset_8600 = 4294967295; BitOffset_8600 = 0; BitLength_8600 = 0; Address_8610 = ''; Type_8610 = ''; AddressPointer_8610 = 0; AdrOffset_8620 = 4294967295; BitOffset_8620 = 0; BitLength_8620 = 0; Address_8620 = ''; Type_8620 = ''; AddressPointer_8620 = 0
    ModbusTCP_Slave_Device : Modbus TCP Slave, Leadshine Technology Co., Ltd., version 00.00.00.10
        settings: SlaveID = 1; portNo = 503
  AC_GENERATOR_DATA
*)

// Device/Application/PLC_PRG
PROGRAM PLC_PRG
VAR
	MC_Power_0: MC_Power;
	MC_Jog_0: MC_Jog;
	MC_MoveRelative_0: MC_MoveRelative;
	MC_Home_0: MC_Home;
	MC_Power_1: MC_Power;
	MC_Jog_1: MC_Jog;
	ix0: BOOL;
	MC_Jog_2: MC_Jog;
	MC_Power_2: MC_Power;
	MC_MoveRelative_1: MC_MoveRelative;
	MC_MoveRelative_2: MC_MoveRelative;
	MC_MoveRelative_3: MC_MoveRelative;
	LS_2AxisLineRel_0: LS_2AxisLineRel;
	pos1: ARRAY [0..2] OF LREAL;
	MC_Home_1: MC_Home;
	MC_Home_2: MC_Home;
	MC_Home_3: MC_Home;
	LS_3AxisLineAbs_0: LS_3AxisLineAbs;
	pos: ARRAY [0..2] OF LREAL;
	done1: BOOL;
	LS_3AxisLineAbs_1: LS_3AxisLineAbs;
	done2: BOOL;
	pos2: ARRAY [0..2] OF LREAL;
	LS_3AxisLineAbs_2: LS_3AxisLineAbs;
	MC_Power_3: MC_Power;
	MC_Home_4: MC_Home;
	MC_MoveAbsolute_0: MC_MoveAbsolute;
	photo_on: INT := 1;
	SMC_GroupPower_0: SMC_GroupPower;
	MC_GroupEnable_0: MC_GroupEnable;
	MC_SetCoordinateTransform_0: MC_SetCoordinateTransform;
	mcs: MC_COORD_REF;
	home_dis: LREAL:=-30;
	MC_Home_5: MC_Home;
	MC_Home_6: MC_Home;
	MC_Home_7: MC_Home;
	y_Red: INT;
	x_Red: INT;
	x_Yellow: INT;
	y_Yellow: INT;
	done3: BOOL;
	done4: BOOL;
	pos3: ARRAY [0..2] OF LREAL;
	MC_MoveAbsolute_1: MC_MoveAbsolute;
	LS_3AxisLineAbs_3: LS_3AxisLineAbs;
	done5: BOOL;
	Delta_X_Yellow: INT;
	Delta_Y_Yellow: INT;
	Delta_pos0: SMC_POS_REF;
	Delta_pos1: SMC_POS_REF;
	MC_MoveDirectAbsolute_0: MC_MoveDirectAbsolute;
	MC_MoveDirectAbsolute_1: MC_MoveDirectAbsolute;
	done6: BOOL;
	MC_MoveDirectAbsolute_2: MC_MoveDirectAbsolute;
	doneDelta: BOOL;
	anquan_pos0: SMC_POS_REF;
	delta_photo_on: INT := 0;
	LS_3AxisLineAbs_4: LS_3AxisLineAbs;
	pos4: ARRAY [0..2] OF LREAL;
	x_Green: INT;
	x_Blue: INT;
	y_Blue: INT;
	y_Green: INT;
	LS_3AxisLineAbs_5: LS_3AxisLineAbs;
	pos5: ARRAY [0..2] OF LREAL;
	LS_3AxisLineAbs_6: LS_3AxisLineAbs;
	done7: BOOL;
	pos6: ARRAY [0..2] OF LREAL;
	done8: BOOL;
	pos7: ARRAY [0..2] OF LREAL;
	done_delta_red: BOOL;
	done_back1: BOOL;
	done_delta_yellow: BOOL;
	LS_3AxisLineAbs_7: LS_3AxisLineAbs;
	Home_1: MC_Home;
	Home_3: MC_Home;
	Home_2: MC_Home;
	done_home: BOOL;
	Delta_X_Red: INT;
	Delta_Y_Red: INT;
	Delta_pos2: SMC_POS_REF;
	MC_MoveDirectAbsolute_3: MC_MoveDirectAbsolute;
	MC_MoveDirectAbsolute_4: MC_MoveDirectAbsolute;
	done_back2: BOOL;
	Delta_pos3: SMC_POS_REF;
	MC_MoveDirectAbsolute_5: MC_MoveDirectAbsolute;
	Delta_X_Blue: INT;
	Delta_X_Green: INT;
	Delta_Y_Green: INT;
	Delta_Y_Blue: INT;
	Delta_pos4: SMC_POS_REF;
	done_delta_blue: BOOL;
	MC_MoveDirectAbsolute_6: MC_MoveDirectAbsolute;
	Delta_pos5: SMC_POS_REF;
	done_back3: BOOL;
	Delta_pos6: SMC_POS_REF;
	done_delta_Green: BOOL;
	MC_MoveDirectAbsolute_7: MC_MoveDirectAbsolute;
	Delta_pos7: SMC_POS_REF;
	MC_MoveDirectAbsolute_8: MC_MoveDirectAbsolute;
	done_back4: BOOL;
	no_photo_delta: BOOL;
	Y_Yellow_orin: INT;
	X_Yellow_orin: INT;
	X_Red_orin: INT;
	Y_Red_orin: INT;
	X_Green_orin: INT;
	Y_Green_orin: INT;
	X_Blue_orin: INT;
	Y_Blue_orin: INT;
END_VAR

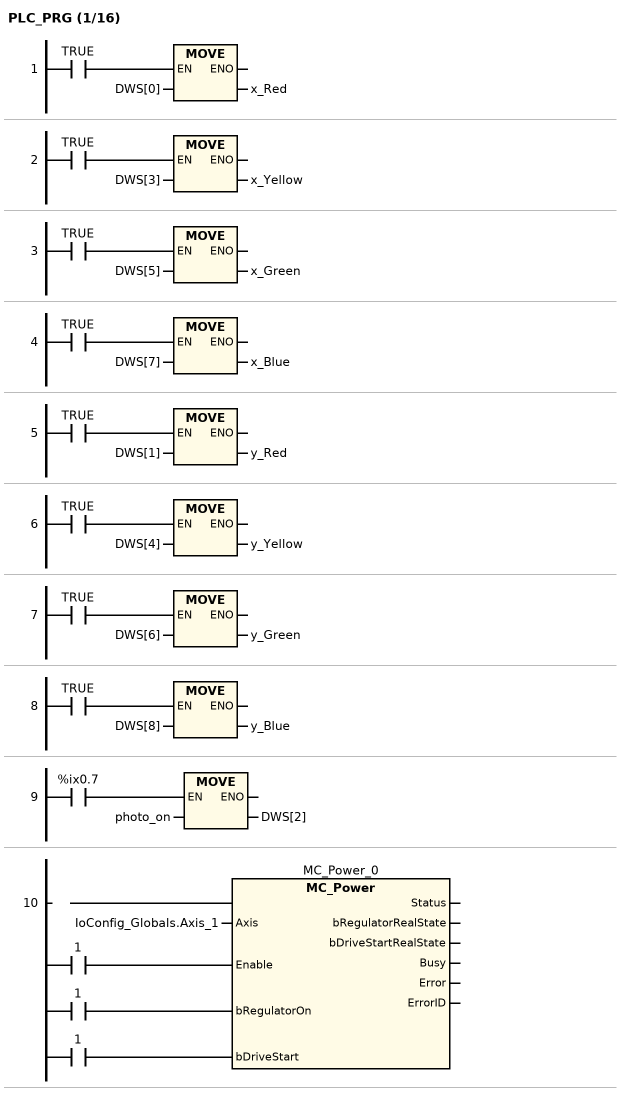
// NETWORK 1
x_Red := DWS[0];

// NETWORK 2
x_Yellow := DWS[3];

// NETWORK 3
x_Green := DWS[5];

// NETWORK 4
x_Blue := DWS[7];

// NETWORK 5
y_Red := DWS[1];

// NETWORK 6
y_Yellow := DWS[4];

// NETWORK 7
y_Green := DWS[6];

// NETWORK 8
y_Blue := DWS[8];

// NETWORK 9
IF %ix0.7 THEN DWS[2] := photo_on; END_IF

// NETWORK 10
MC_Power_0(Axis := IoConfig_Globals.Axis_1, Enable := 1, bRegulatorOn := 1, bDriveStart := 1); // MC_Power

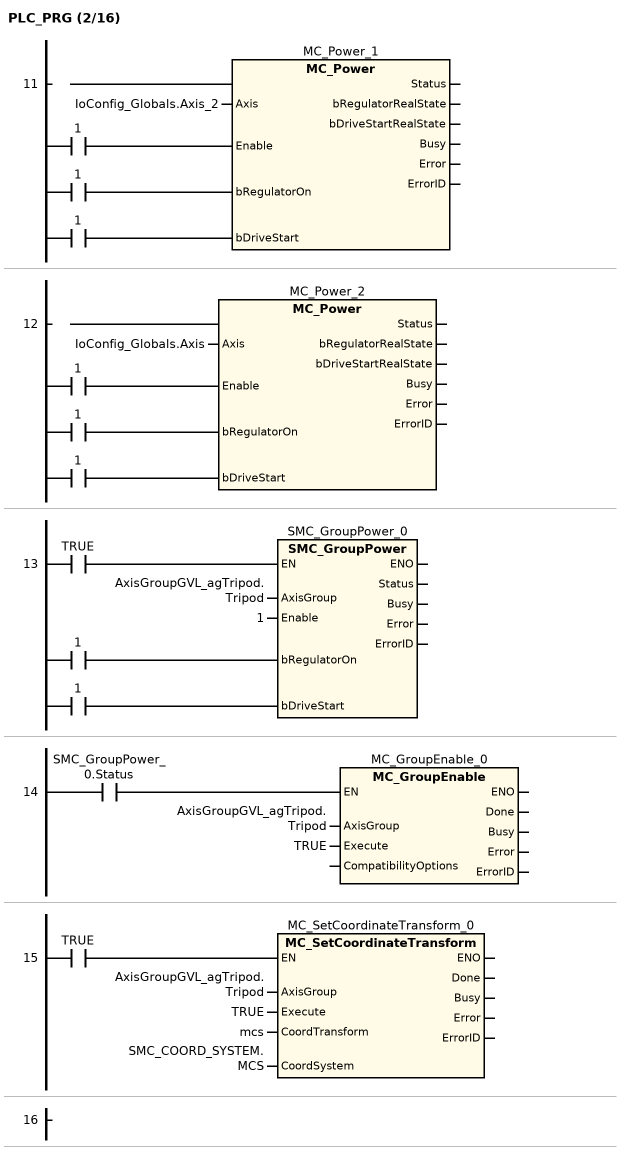
// NETWORK 11
MC_Power_1(Axis := IoConfig_Globals.Axis_2, Enable := 1, bRegulatorOn := 1, bDriveStart := 1); // MC_Power

// NETWORK 12
MC_Power_2(Axis := IoConfig_Globals.Axis, Enable := 1, bRegulatorOn := 1, bDriveStart := 1); // MC_Power

// NETWORK 13
SMC_GroupPower_0(AxisGroup := AxisGroupGVL_agTripod.Tripod, Enable := 1, bRegulatorOn := 1, bDriveStart := 1); // SMC_GroupPower

// NETWORK 14
IF SMC_GroupPower_0.Status THEN
    MC_GroupEnable_0(AxisGroup := AxisGroupGVL_agTripod.Tripod, Execute := TRUE); // MC_GroupEnable
END_IF

// NETWORK 15
MC_SetCoordinateTransform_0(
    AxisGroup := AxisGroupGVL_agTripod.Tripod,
    Execute := TRUE,
    CoordTransform := mcs,
    CoordSystem := SMC_COORD_SYSTEM.MCS); // MC_SetCoordinateTransform

// NETWORK 16

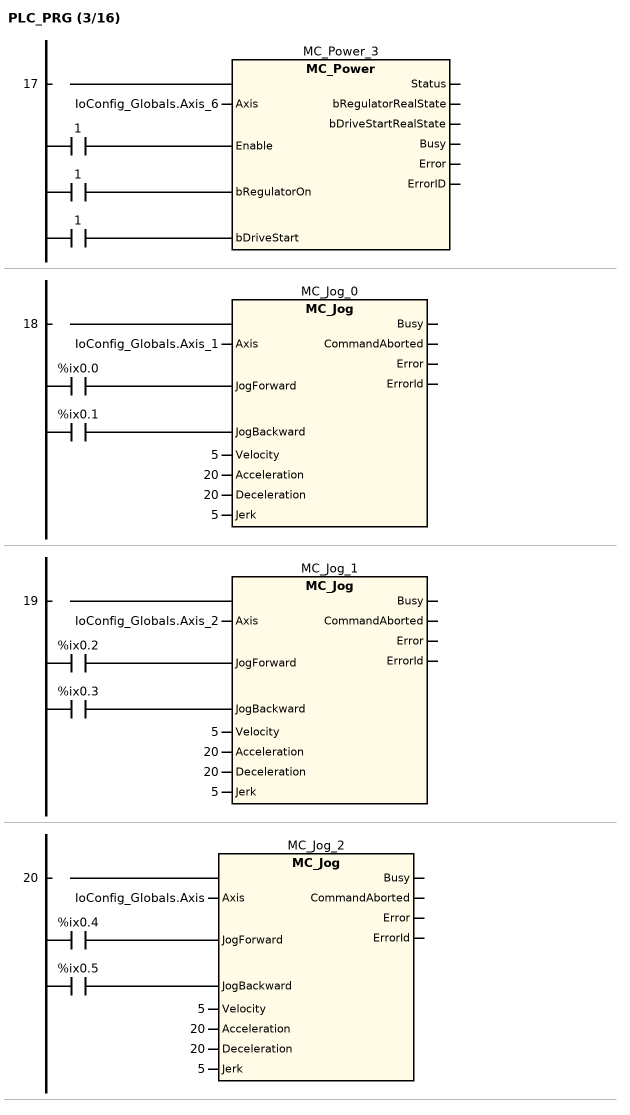
// NETWORK 17
MC_Power_3(Axis := IoConfig_Globals.Axis_6, Enable := 1, bRegulatorOn := 1, bDriveStart := 1); // MC_Power

// NETWORK 18
MC_Jog_0(
    Axis := IoConfig_Globals.Axis_1,
    JogForward := %ix0.0,
    JogBackward := %ix0.1,
    Velocity := 5,
    Acceleration := 20,
    Deceleration := 20,
    Jerk := 5); // MC_Jog

// NETWORK 19
MC_Jog_1(
    Axis := IoConfig_Globals.Axis_2,
    JogForward := %ix0.2,
    JogBackward := %ix0.3,
    Velocity := 5,
    Acceleration := 20,
    Deceleration := 20,
    Jerk := 5); // MC_Jog

// NETWORK 20
MC_Jog_2(
    Axis := IoConfig_Globals.Axis,
    JogForward := %ix0.4,
    JogBackward := %ix0.5,
    Velocity := 5,
    Acceleration := 20,
    Deceleration := 20,
    Jerk := 5); // MC_Jog

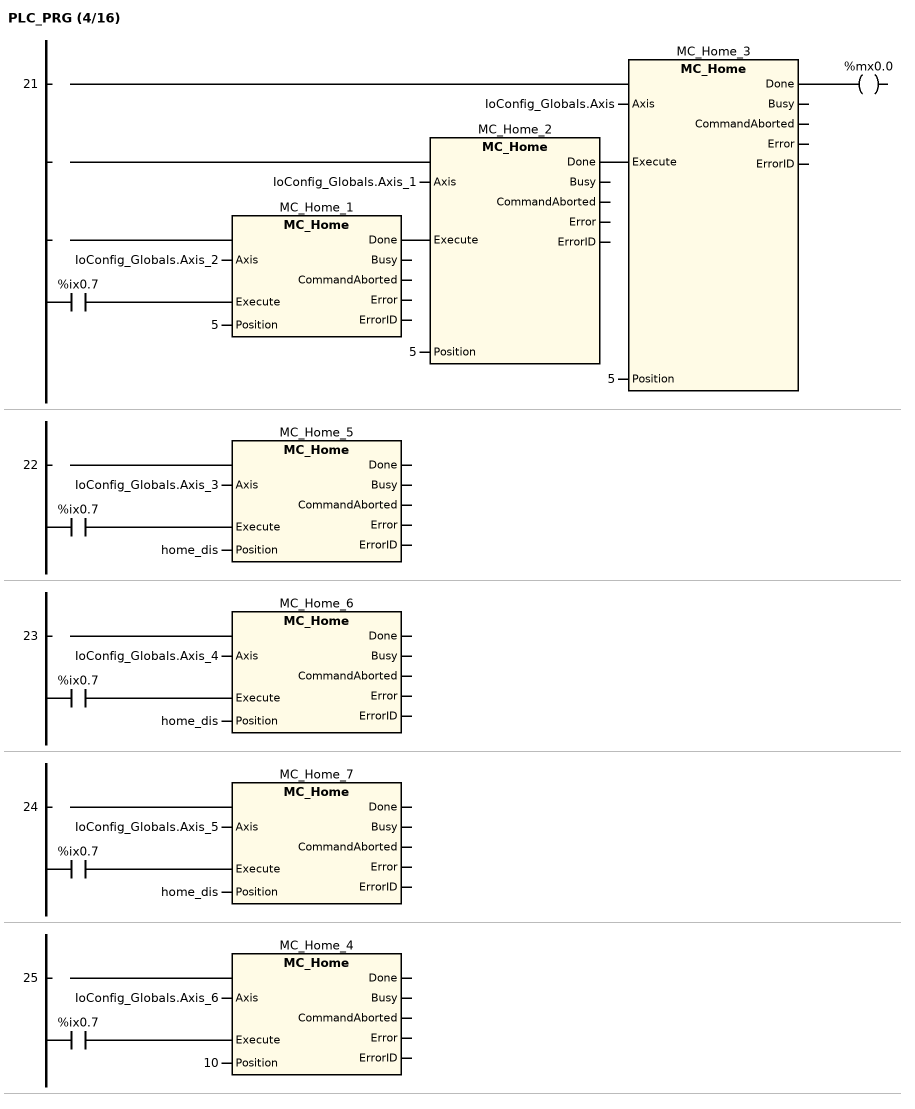
// NETWORK 21
MC_Home_1(Axis := IoConfig_Globals.Axis_2, Execute := %ix0.7, Position := 5); // MC_Home
MC_Home_2(Axis := IoConfig_Globals.Axis_1, Execute := MC_Home_1.Done, Position := 5); // MC_Home
MC_Home_3(Axis := IoConfig_Globals.Axis, Execute := MC_Home_2.Done, Position := 5); // MC_Home
%mx0.0 := MC_Home_3.Done;

// NETWORK 22
MC_Home_5(Axis := IoConfig_Globals.Axis_3, Execute := %ix0.7, Position := home_dis); // MC_Home

// NETWORK 23
MC_Home_6(Axis := IoConfig_Globals.Axis_4, Execute := %ix0.7, Position := home_dis); // MC_Home

// NETWORK 24
MC_Home_7(Axis := IoConfig_Globals.Axis_5, Execute := %ix0.7, Position := home_dis); // MC_Home

// NETWORK 25
MC_Home_4(Axis := IoConfig_Globals.Axis_6, Execute := %ix0.7, Position := 10); // MC_Home

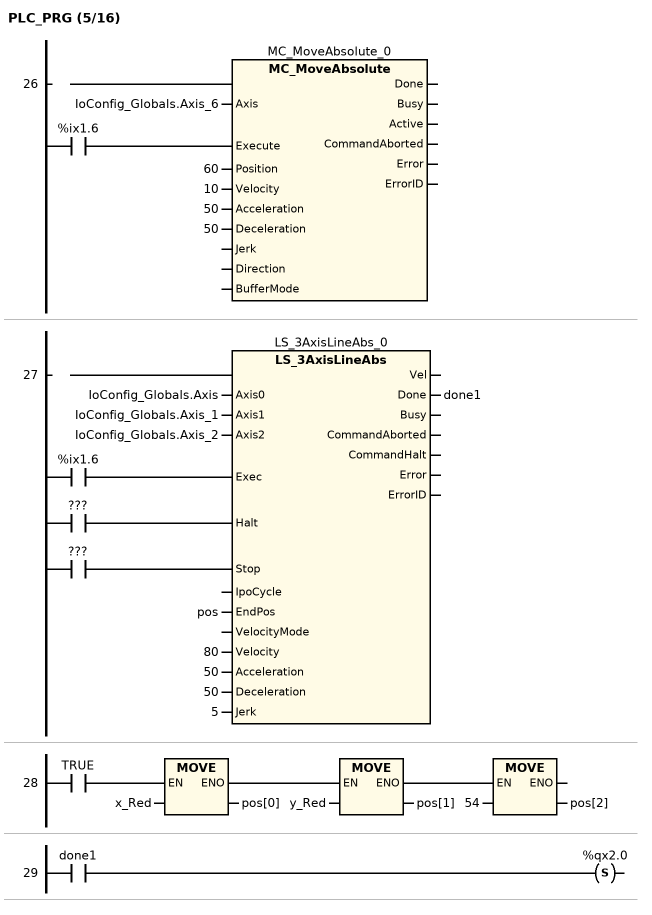
// NETWORK 26
MC_MoveAbsolute_0(
    Axis := IoConfig_Globals.Axis_6,
    Execute := %ix1.6,
    Position := 60,
    Velocity := 10,
    Acceleration := 50,
    Deceleration := 50); // MC_MoveAbsolute

// NETWORK 27
LS_3AxisLineAbs_0(
    Axis0 := IoConfig_Globals.Axis,
    Axis1 := IoConfig_Globals.Axis_1,
    Axis2 := IoConfig_Globals.Axis_2,
    Exec := %ix1.6,
    EndPos := pos,
    Velocity := 80,
    Acceleration := 50,
    Deceleration := 50,
    Jerk := 5,
    Done => done1); // LS_3AxisLineAbs

// NETWORK 28
pos[0] := x_Red;
pos[1] := y_Red;
pos[2] := 54;

// NETWORK 29
%qx2.0 S= done1;

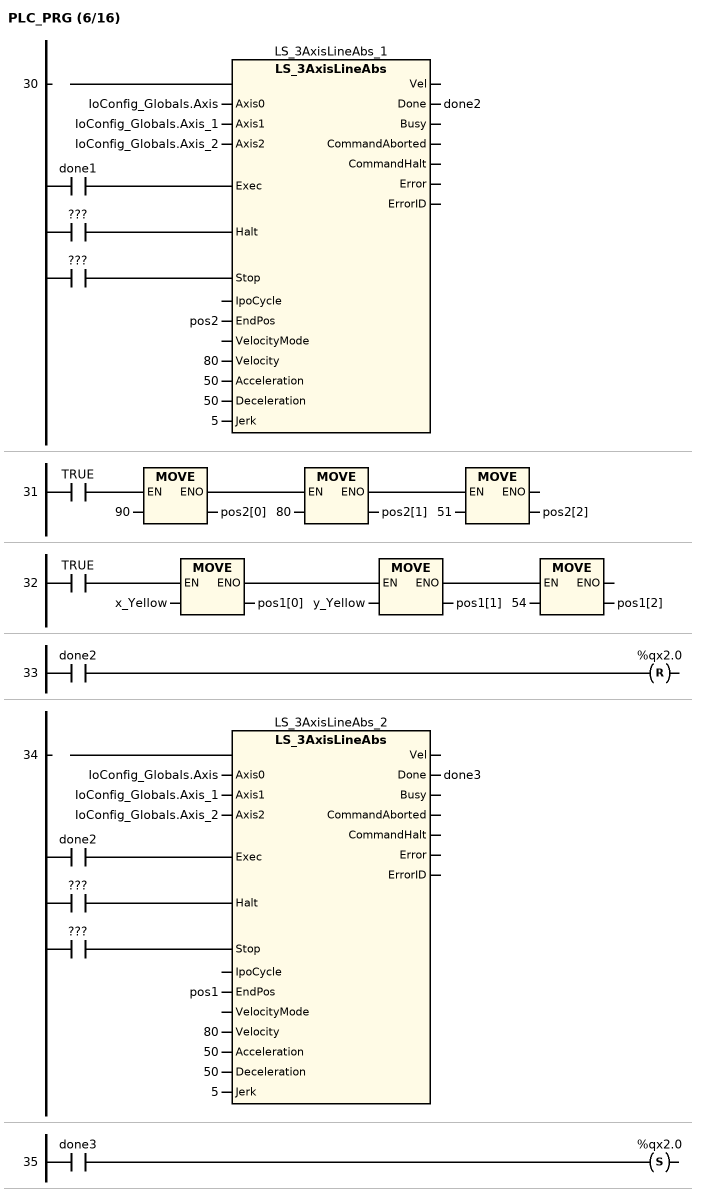
// NETWORK 30
LS_3AxisLineAbs_1(
    Axis0 := IoConfig_Globals.Axis,
    Axis1 := IoConfig_Globals.Axis_1,
    Axis2 := IoConfig_Globals.Axis_2,
    Exec := done1,
    EndPos := pos2,
    Velocity := 80,
    Acceleration := 50,
    Deceleration := 50,
    Jerk := 5,
    Done => done2); // LS_3AxisLineAbs

// NETWORK 31
pos2[0] := 90;
pos2[1] := 80;
pos2[2] := 51;

// NETWORK 32
pos1[0] := x_Yellow;
pos1[1] := y_Yellow;
pos1[2] := 54;

// NETWORK 33
%qx2.0 R= done2;

// NETWORK 34
LS_3AxisLineAbs_2(
    Axis0 := IoConfig_Globals.Axis,
    Axis1 := IoConfig_Globals.Axis_1,
    Axis2 := IoConfig_Globals.Axis_2,
    Exec := done2,
    EndPos := pos1,
    Velocity := 80,
    Acceleration := 50,
    Deceleration := 50,
    Jerk := 5,
    Done => done3); // LS_3AxisLineAbs

// NETWORK 35
%qx2.0 S= done3;

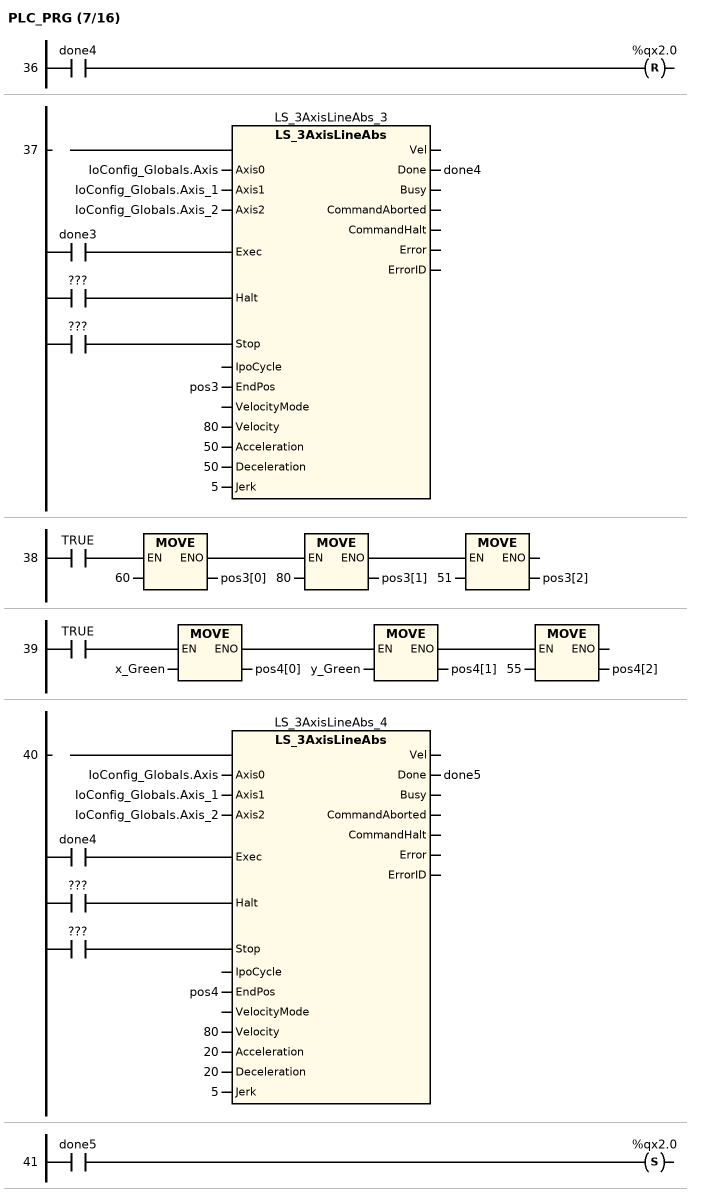
// NETWORK 36
%qx2.0 R= done4;

// NETWORK 37
LS_3AxisLineAbs_3(
    Axis0 := IoConfig_Globals.Axis,
    Axis1 := IoConfig_Globals.Axis_1,
    Axis2 := IoConfig_Globals.Axis_2,
    Exec := done3,
    EndPos := pos3,
    Velocity := 80,
    Acceleration := 50,
    Deceleration := 50,
    Jerk := 5,
    Done => done4); // LS_3AxisLineAbs

// NETWORK 38
pos3[0] := 60;
pos3[1] := 80;
pos3[2] := 51;

// NETWORK 39
pos4[0] := x_Green;
pos4[1] := y_Green;
pos4[2] := 55;

// NETWORK 40
LS_3AxisLineAbs_4(
    Axis0 := IoConfig_Globals.Axis,
    Axis1 := IoConfig_Globals.Axis_1,
    Axis2 := IoConfig_Globals.Axis_2,
    Exec := done4,
    EndPos := pos4,
    Velocity := 80,
    Acceleration := 20,
    Deceleration := 20,
    Jerk := 5,
    Done => done5); // LS_3AxisLineAbs

// NETWORK 41
%qx2.0 S= done5;

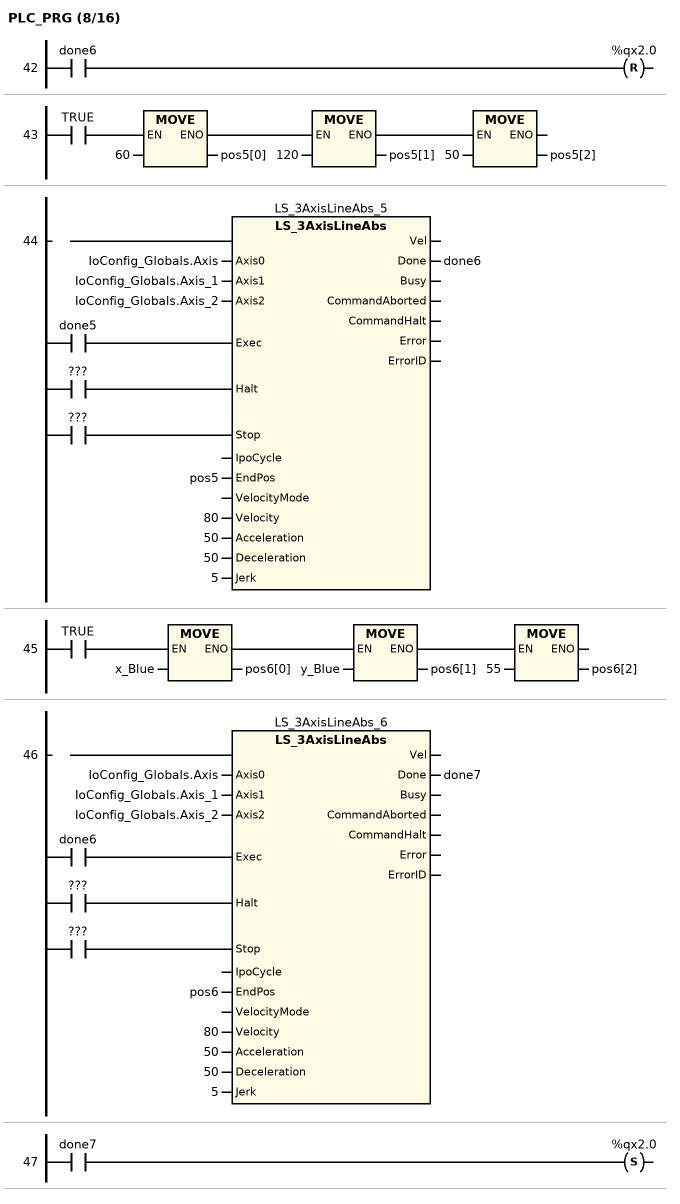
// NETWORK 42
%qx2.0 R= done6;

// NETWORK 43
pos5[0] := 60;
pos5[1] := 120;
pos5[2] := 50;

// NETWORK 44
LS_3AxisLineAbs_5(
    Axis0 := IoConfig_Globals.Axis,
    Axis1 := IoConfig_Globals.Axis_1,
    Axis2 := IoConfig_Globals.Axis_2,
    Exec := done5,
    EndPos := pos5,
    Velocity := 80,
    Acceleration := 50,
    Deceleration := 50,
    Jerk := 5,
    Done => done6); // LS_3AxisLineAbs

// NETWORK 45
pos6[0] := x_Blue;
pos6[1] := y_Blue;
pos6[2] := 55;

// NETWORK 46
LS_3AxisLineAbs_6(
    Axis0 := IoConfig_Globals.Axis,
    Axis1 := IoConfig_Globals.Axis_1,
    Axis2 := IoConfig_Globals.Axis_2,
    Exec := done6,
    EndPos := pos6,
    Velocity := 80,
    Acceleration := 50,
    Deceleration := 50,
    Jerk := 5,
    Done => done7); // LS_3AxisLineAbs

// NETWORK 47
%qx2.0 S= done7;

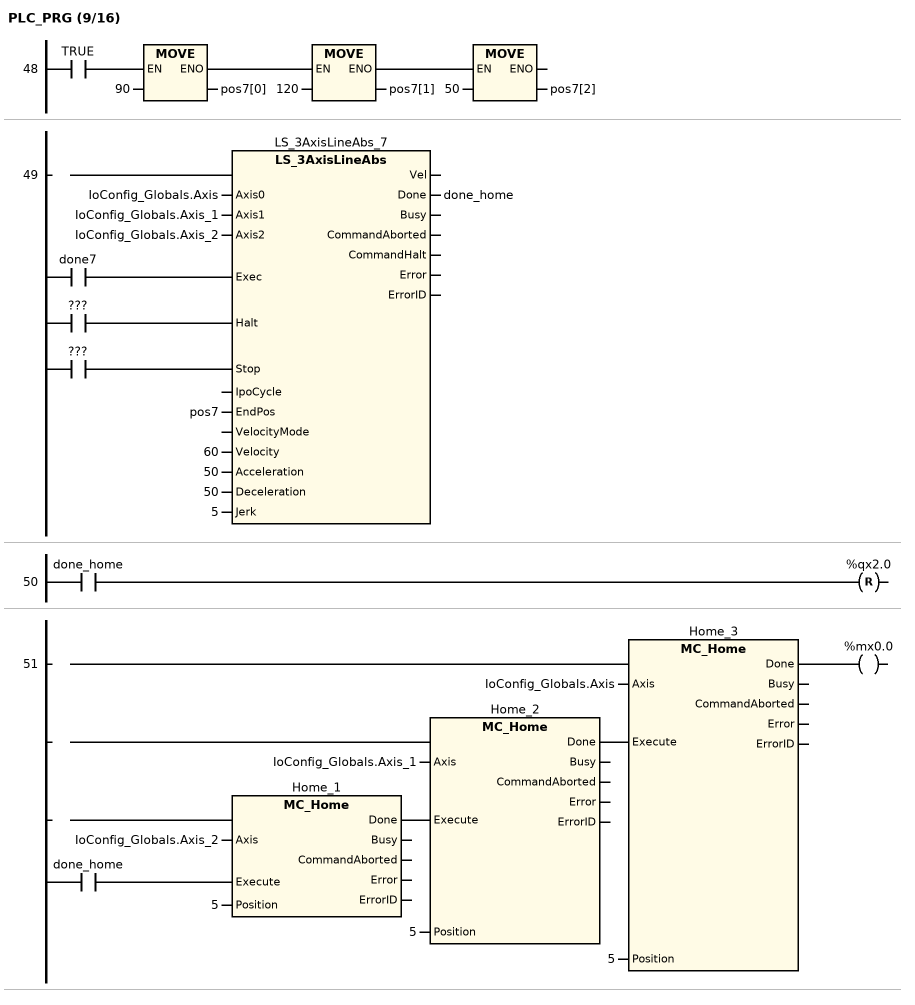
// NETWORK 48
pos7[0] := 90;
pos7[1] := 120;
pos7[2] := 50;

// NETWORK 49
LS_3AxisLineAbs_7(
    Axis0 := IoConfig_Globals.Axis,
    Axis1 := IoConfig_Globals.Axis_1,
    Axis2 := IoConfig_Globals.Axis_2,
    Exec := done7,
    EndPos := pos7,
    Velocity := 60,
    Acceleration := 50,
    Deceleration := 50,
    Jerk := 5,
    Done => done_home); // LS_3AxisLineAbs

// NETWORK 50
%qx2.0 R= done_home;

// NETWORK 51
Home_1(Axis := IoConfig_Globals.Axis_2, Execute := done_home, Position := 5); // MC_Home
Home_2(Axis := IoConfig_Globals.Axis_1, Execute := Home_1.Done, Position := 5); // MC_Home
Home_3(Axis := IoConfig_Globals.Axis, Execute := Home_2.Done, Position := 5); // MC_Home
%mx0.0 := Home_3.Done;

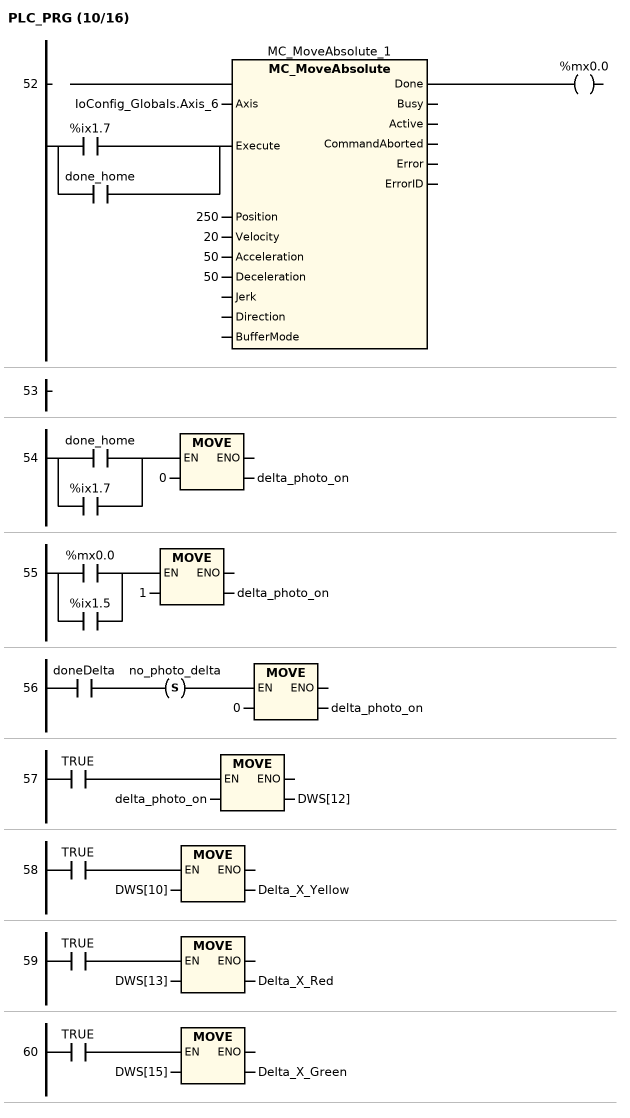
// NETWORK 52
MC_MoveAbsolute_1(
    Axis := IoConfig_Globals.Axis_6,
    Execute := %ix1.7 OR done_home,
    Position := 250,
    Velocity := 20,
    Acceleration := 50,
    Deceleration := 50); // MC_MoveAbsolute
%mx0.0 := MC_MoveAbsolute_1.Done;

// NETWORK 53

// NETWORK 54
IF done_home OR %ix1.7 THEN delta_photo_on := 0; END_IF

// NETWORK 55
IF %mx0.0 OR %ix1.5 THEN delta_photo_on := 1; END_IF

// NETWORK 56
no_photo_delta S= doneDelta;
IF doneDelta THEN delta_photo_on := 0; END_IF

// NETWORK 57
DWS[12] := delta_photo_on;

// NETWORK 58
Delta_X_Yellow := DWS[10];

// NETWORK 59
Delta_X_Red := DWS[13];

// NETWORK 60
Delta_X_Green := DWS[15];

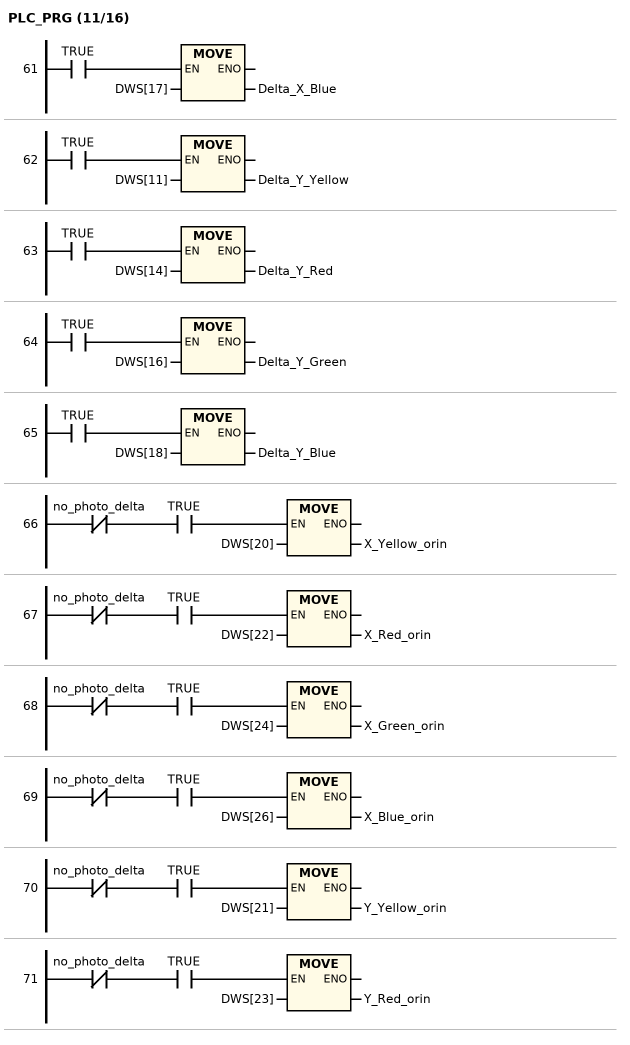
// NETWORK 61
Delta_X_Blue := DWS[17];

// NETWORK 62
Delta_Y_Yellow := DWS[11];

// NETWORK 63
Delta_Y_Red := DWS[14];

// NETWORK 64
Delta_Y_Green := DWS[16];

// NETWORK 65
Delta_Y_Blue := DWS[18];

// NETWORK 66
IF NOT no_photo_delta AND TRUE THEN X_Yellow_orin := DWS[20]; END_IF

// NETWORK 67
IF NOT no_photo_delta AND TRUE THEN X_Red_orin := DWS[22]; END_IF

// NETWORK 68
IF NOT no_photo_delta AND TRUE THEN X_Green_orin := DWS[24]; END_IF

// NETWORK 69
IF NOT no_photo_delta AND TRUE THEN X_Blue_orin := DWS[26]; END_IF

// NETWORK 70
IF NOT no_photo_delta AND TRUE THEN Y_Yellow_orin := DWS[21]; END_IF

// NETWORK 71
IF NOT no_photo_delta AND TRUE THEN Y_Red_orin := DWS[23]; END_IF

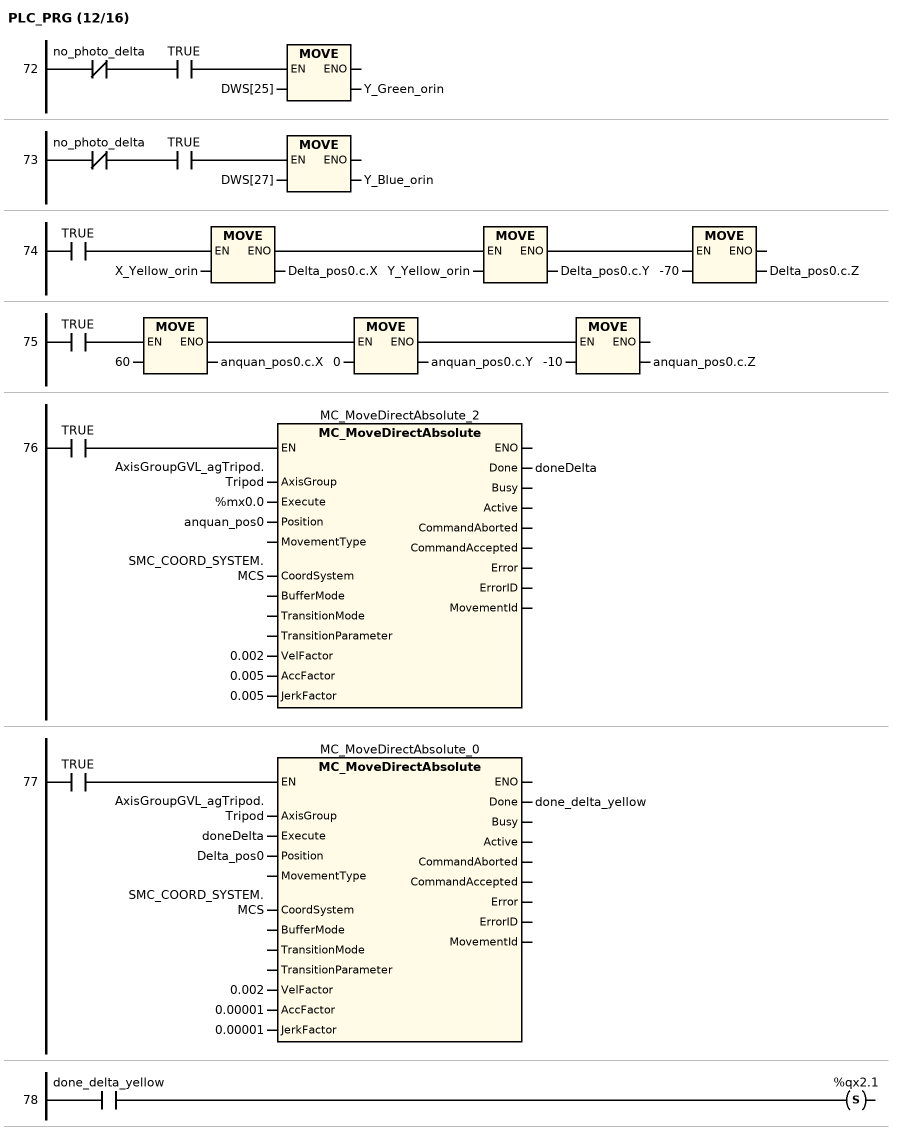
// NETWORK 72
IF NOT no_photo_delta AND TRUE THEN Y_Green_orin := DWS[25]; END_IF

// NETWORK 73
IF NOT no_photo_delta AND TRUE THEN Y_Blue_orin := DWS[27]; END_IF

// NETWORK 74
Delta_pos0.c.X := X_Yellow_orin;
Delta_pos0.c.Y := Y_Yellow_orin;
Delta_pos0.c.Z := -70;

// NETWORK 75
anquan_pos0.c.X := 60;
anquan_pos0.c.Y := 0;
anquan_pos0.c.Z := -10;

// NETWORK 76
MC_MoveDirectAbsolute_2(
    AxisGroup := AxisGroupGVL_agTripod.Tripod,
    Execute := %mx0.0,
    Position := anquan_pos0,
    CoordSystem := SMC_COORD_SYSTEM.MCS,
    VelFactor := 0.002,
    AccFactor := 0.005,
    JerkFactor := 0.005,
    Done => doneDelta); // MC_MoveDirectAbsolute

// NETWORK 77
MC_MoveDirectAbsolute_0(
    AxisGroup := AxisGroupGVL_agTripod.Tripod,
    Execute := doneDelta,
    Position := Delta_pos0,
    CoordSystem := SMC_COORD_SYSTEM.MCS,
    VelFactor := 0.002,
    AccFactor := 0.00001,
    JerkFactor := 0.00001,
    Done => done_delta_yellow); // MC_MoveDirectAbsolute

// NETWORK 78
%qx2.1 S= done_delta_yellow;

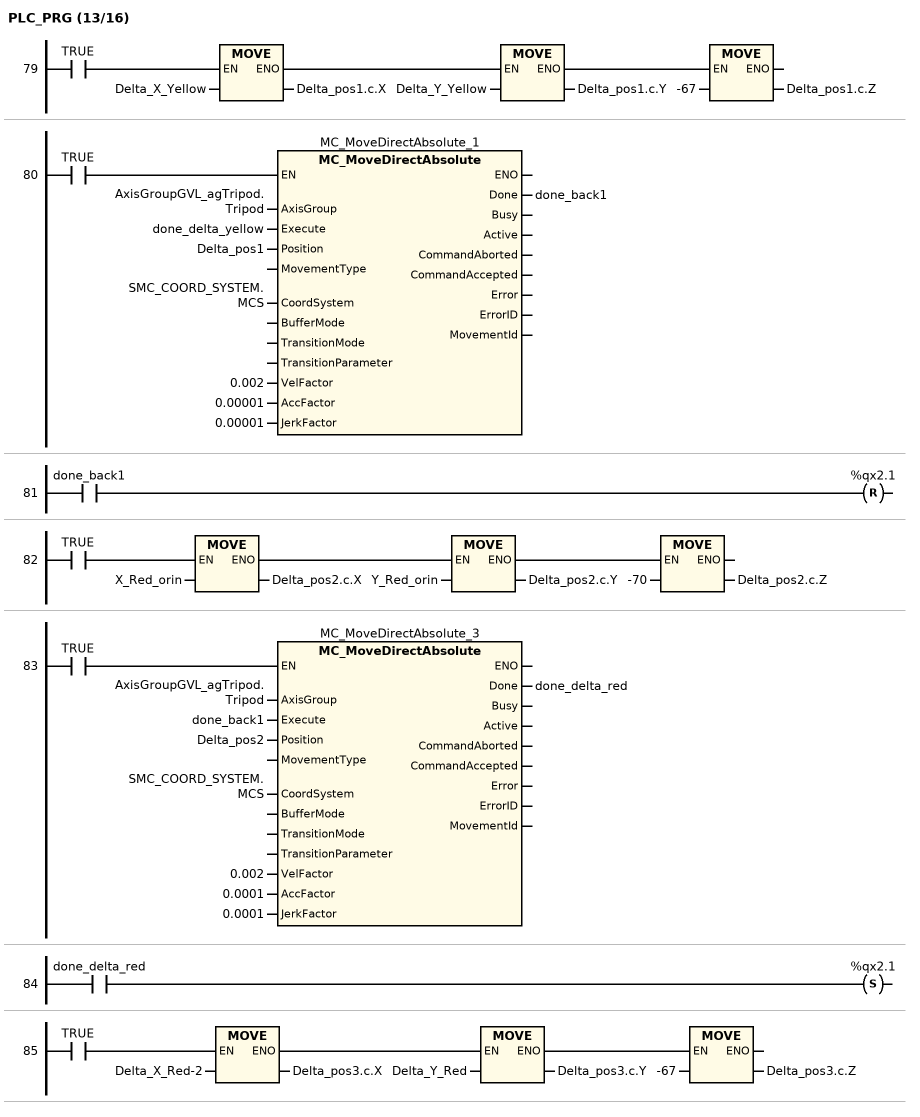
// NETWORK 79
Delta_pos1.c.X := Delta_X_Yellow;
Delta_pos1.c.Y := Delta_Y_Yellow;
Delta_pos1.c.Z := -67;

// NETWORK 80
MC_MoveDirectAbsolute_1(
    AxisGroup := AxisGroupGVL_agTripod.Tripod,
    Execute := done_delta_yellow,
    Position := Delta_pos1,
    CoordSystem := SMC_COORD_SYSTEM.MCS,
    VelFactor := 0.002,
    AccFactor := 0.00001,
    JerkFactor := 0.00001,
    Done => done_back1); // MC_MoveDirectAbsolute

// NETWORK 81
%qx2.1 R= done_back1;

// NETWORK 82
Delta_pos2.c.X := X_Red_orin;
Delta_pos2.c.Y := Y_Red_orin;
Delta_pos2.c.Z := -70;

// NETWORK 83
MC_MoveDirectAbsolute_3(
    AxisGroup := AxisGroupGVL_agTripod.Tripod,
    Execute := done_back1,
    Position := Delta_pos2,
    CoordSystem := SMC_COORD_SYSTEM.MCS,
    VelFactor := 0.002,
    AccFactor := 0.0001,
    JerkFactor := 0.0001,
    Done => done_delta_red); // MC_MoveDirectAbsolute

// NETWORK 84
%qx2.1 S= done_delta_red;

// NETWORK 85
Delta_pos3.c.X := Delta_X_Red-2;
Delta_pos3.c.Y := Delta_Y_Red;
Delta_pos3.c.Z := -67;

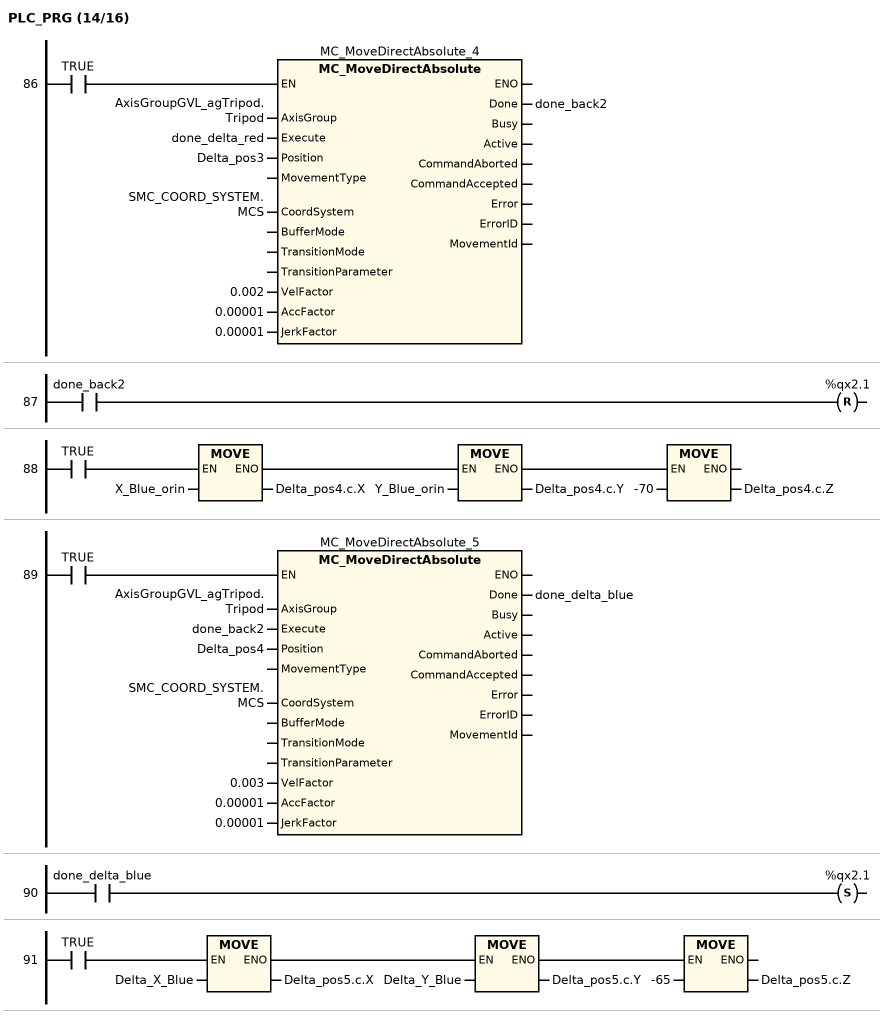
// NETWORK 86
MC_MoveDirectAbsolute_4(
    AxisGroup := AxisGroupGVL_agTripod.Tripod,
    Execute := done_delta_red,
    Position := Delta_pos3,
    CoordSystem := SMC_COORD_SYSTEM.MCS,
    VelFactor := 0.002,
    AccFactor := 0.00001,
    JerkFactor := 0.00001,
    Done => done_back2); // MC_MoveDirectAbsolute

// NETWORK 87
%qx2.1 R= done_back2;

// NETWORK 88
Delta_pos4.c.X := X_Blue_orin;
Delta_pos4.c.Y := Y_Blue_orin;
Delta_pos4.c.Z := -70;

// NETWORK 89
MC_MoveDirectAbsolute_5(
    AxisGroup := AxisGroupGVL_agTripod.Tripod,
    Execute := done_back2,
    Position := Delta_pos4,
    CoordSystem := SMC_COORD_SYSTEM.MCS,
    VelFactor := 0.003,
    AccFactor := 0.00001,
    JerkFactor := 0.00001,
    Done => done_delta_blue); // MC_MoveDirectAbsolute

// NETWORK 90
%qx2.1 S= done_delta_blue;

// NETWORK 91
Delta_pos5.c.X := Delta_X_Blue;
Delta_pos5.c.Y := Delta_Y_Blue;
Delta_pos5.c.Z := -65;

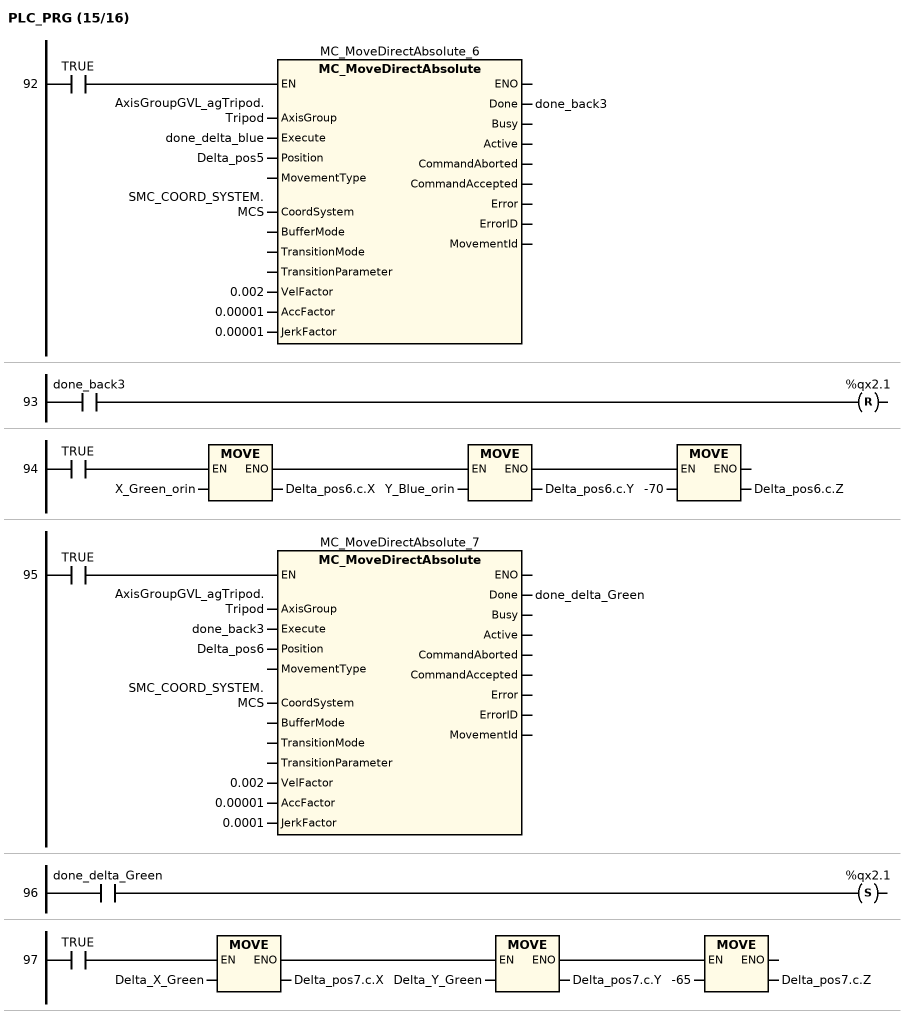
// NETWORK 92
MC_MoveDirectAbsolute_6(
    AxisGroup := AxisGroupGVL_agTripod.Tripod,
    Execute := done_delta_blue,
    Position := Delta_pos5,
    CoordSystem := SMC_COORD_SYSTEM.MCS,
    VelFactor := 0.002,
    AccFactor := 0.00001,
    JerkFactor := 0.00001,
    Done => done_back3); // MC_MoveDirectAbsolute

// NETWORK 93
%qx2.1 R= done_back3;

// NETWORK 94
Delta_pos6.c.X := X_Green_orin;
Delta_pos6.c.Y := Y_Blue_orin;
Delta_pos6.c.Z := -70;

// NETWORK 95
MC_MoveDirectAbsolute_7(
    AxisGroup := AxisGroupGVL_agTripod.Tripod,
    Execute := done_back3,
    Position := Delta_pos6,
    CoordSystem := SMC_COORD_SYSTEM.MCS,
    VelFactor := 0.002,
    AccFactor := 0.00001,
    JerkFactor := 0.0001,
    Done => done_delta_Green); // MC_MoveDirectAbsolute

// NETWORK 96
%qx2.1 S= done_delta_Green;

// NETWORK 97
Delta_pos7.c.X := Delta_X_Green;
Delta_pos7.c.Y := Delta_Y_Green;
Delta_pos7.c.Z := -65;

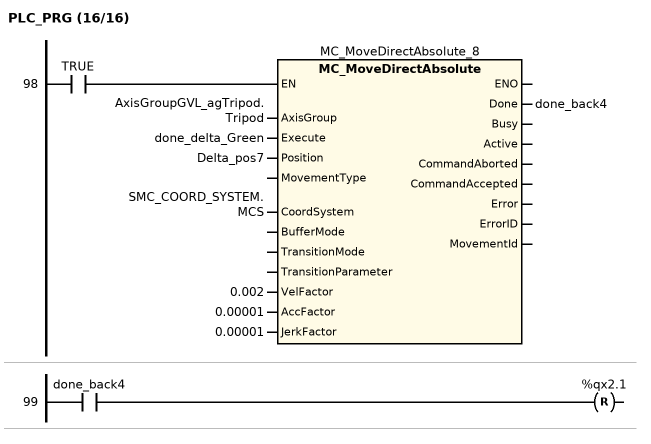
// NETWORK 98
MC_MoveDirectAbsolute_8(
    AxisGroup := AxisGroupGVL_agTripod.Tripod,
    Execute := done_delta_Green,
    Position := Delta_pos7,
    CoordSystem := SMC_COORD_SYSTEM.MCS,
    VelFactor := 0.002,
    AccFactor := 0.00001,
    JerkFactor := 0.00001,
    Done => done_back4); // MC_MoveDirectAbsolute

// NETWORK 99
%qx2.1 R= done_back4;

END_PROGRAM
